// TIA Portal V20 export
// export: Created 2025-12-01T14:57:40.422597Z, ExportSetting None, DisplayName Totally Integrated Automation Portal, DisplayVersion V20 Update 3, DisplayName TIA Portal Openness, DisplayVersion V20 Update 3, DisplayName TIA Portal Version Control Interface, DisplayVersion V20 Update 3, DisplayName STEP 7 Professional, DisplayVersion V20 Update 3, DisplayName STEP 7 Safety, DisplayVersion V20 Update 2, DisplayName WinCC Basic/Comfort/Advanced, DisplayVersion V20 Update 3, DisplayName WinCC Professional, DisplayVersion V20 Update 3, DisplayName WinCC Unified, DisplayVersion V20 Update 3
FUNCTION_BLOCK "FB290_M_CIMCORP_Carga"   // FB290, LAD
TITLE = M_TRANSLO_CS_CARGA_E1_S0
{ S7_Optimized_Access := 'FALSE' }
AUTHOR : CIMCORP
NAME : 20170822
VERSION : 3.5
// stored: AutoNumber false, SetENOAutomatically false
   VAR_INPUT
      Mesa : UInt;   // Mesa de la FB
      Error_Tx : Bool;   // Error en el Tx
      EnTension : Bool;   // Existe Tension en la Mesa
      Termico_Tx : Bool;   // Proteccion del Tx
      pHsMx_1 : Bool;   // pHs 1 de la Mesa
      pHsMx_2 : Bool;   // pHs 2 de la Mesa
      pHsMx_Seg : Bool;   // pHs Seguridad de la Mesa
      Avance_Tx : Bool;   // Avance del Tx
      CIMCORP_MoveOK : Bool;   // CIMCORP >> Move OK
      CIMCORP_Stop : Bool;   // CIMCORP >> Stop
      Centrador_OUT : Bool;   // CENTRADOR >> OUT - Fuera
      Centrador_IN { ExternalAccessible := 'False'; ExternalVisible := 'False'; ExternalWritable := 'False'} : Bool;   // CENTRADOR >> IN - Dentro
      Centrador_EnMovimiento : Bool;   // CENTRADOR >> En Movimiento
      MAnt_CajaPequena : Bool;   // E1 >> Mesa Anterior Caja Pequeña
      MAnt_DescargaAct : Bool;   // E1 >> Mesa Anterior DescargaAct
      AVTF_MAnt_Mx : Bool;   // E1 >> Mesa Anterior AVTF
      P_Mens_MAnt_Mx : Bool;   // E1 >> Mesa Anterior P_Mens
      Mx_ControlUTs : Bool;   // Config >> Control de UT en Mesa
      Mx_VelocidadLenta_In : Bool;   // Forzar a Velociada Lenta
      F_EnvMens_Mx : Bool;   // Fin de Envio de Mensaje
      OrdSal_S00 : Bool;   // Orden de Salida por S0
      V_CNT_pHsMx : Int := 400;   // Valor de Presencia
      V_CNTSeg_pHsMx : Int := 2000;   // Valor de Seguriadad para Presencia
      V_CNT_PasoLenta : Int := 2000;   // Valor de Paso a Lenta
      V_TOut_Tx_Mx : Int := 15000;   // TimeOut de Entrada por E1
      V_TOut_Centrador : Int := 5000;   // TimeOut del Centrador
      V_TOut_Horquillado : Int := 10000;   // TimeOut de Horquillado
      V_CNT_PerdidapHs : Int := 1000;   // CNT de Perdida de pHs
      V_CNT_Posicionado : Int := 1000;   // CNT de Posicionado Simple
      V_CNT_CargaCompactada : Int := 1000;   // CNT de Carga Compactada
   END_VAR
   VAR_OUTPUT
      P_EnvMens_PMx : Bool;   // Permiso de Enviar Mensaje de Presencia
      P_EnvMens_AMx : Bool;   // Permiso de Enviar Mensaje de Ausencia
      P_RecepOK_Mx : Bool;   // Recepcion OK
      PTF_MAnt_Mx : Bool;   // E1 >> Mesa Anterior PTF
      FTF_MAnt_Mx : Bool;   // E1 >> Mesa Anterior FTF
   END_VAR
   VAR
      Mx_ET00 : Bool;
      Mx_ET01 : Bool;
      Mx_ET02 : Bool;
      Mx_ET07_1PRE : Bool;
      Mx_ET07_1FIN : Bool;
      Mx_ET07_2PRE : Bool;
      Mx_ET07_2FIN : Bool;
      Mx_ET08 : Bool;
      Mx_ET09 : Bool;
      Mx_ET10Previo : Bool;
      Mx_ET10 : Bool;
      Mx_ET11 : Bool;
      Mx_ET12 : Bool;
      Mx_ET110 : Bool;
      Mx_ET111 : Bool;
      Mx_ET02ESPERA : Bool;
      Mx_ET50 : Bool;
      Mx_ET51 : Bool;
      Mx_ET52 : Bool;
      MX_ET150 : Bool;
      Mx_ET151 : Bool;
      Mx_EnResetDoblePres : Bool;   // Config >> En Reset Doble Presencia
      CIMCORP_OK : Bool;   // CIMCORP >> Esta En Marcha
      SinUTs_EnMesa : Bool;   // Control UTs En Mesa >> Sin UTs
      DoblePeque_EnMesa : Bool;   // Control UTs En Mesa >> Caja Doble Pequeña
      UT01Peque_EnMesa : Bool;   // Control UTs En Mesa >> UT01 Caja Pequeña
      UT02Peque_EnMesa : Bool;   // Control UTs En Mesa >> UT02 Caja Pequeña
      OrdSalida_OK : Bool;   // Control UTs En Mesa >> Validar Orden de Salida
      EntrandoDobleCaja : Bool;   // Interna >> Entrando Doble Caja
      SalidaDobleCaja : Bool;   // Interna >> Salida de Caja Grande o Dos Pequeñas
      SalidaSimpleCaja : Bool;   // Interna >> Salida de Caja pequeña
      CargaCompactada : Bool;   // Interna >> Carga Compactada
      MemoriaCentrador_IN : Bool;   // Interna >> Memoria para la Señal de Centrador IN
      ProtocoloIniciado : Bool;   // Iniciado el Envio del Mensaje de Presencia
      CNT_pHsMx { S7_SetPoint := 'True'} : "FB910_CNT_UHS";   // CNT de la Presencia
      CNTSeg_pHsMx { S7_SetPoint := 'True'} : "FB910_CNT_UHS";   // CNT de Seguridad de la Presencia
      TMP_EnTension { S7_SetPoint := 'True'} : "FB910_CNT_UHS";
      TOut_Av_Tx { ExternalWritable := 'False'; S7_SetPoint := 'True'} : "FB910_CNT_UHS";   // Time Out de Entrada de E1
      TOut_SacarCentrador { S7_SetPoint := 'True'} : "FB910_CNT_UHS";
      TOut_RecogerCentrador { S7_SetPoint := 'True'} : "FB910_CNT_UHS";
      TOut_Horquillado { S7_SetPoint := 'True'} : "FB910_CNT_UHS";
      CNT_PerdidapHs { S7_SetPoint := 'True'} : "FB910_CNT_UHS";   // CNT de Perdida de pHs
      CNT_Posicionado { S7_SetPoint := 'True'} : "FB910_CNT_UHS";   // CNT de Posicionado Simple
      CNT_CargaCompactada { S7_SetPoint := 'True'} : "FB910_CNT_UHS";   // CNT de Carga Compactada
      STAT_EnvMens_PMx : Bool;   // Interna >> Envio del Mensaje de Presencia
      STAT_EnvMens_AMx : Bool;   // Interna >> Envio de Mensaje de Ausencia
      STAT_FTF_MAnt_Mx : Bool;   // Interna >> FTF de MAnt >> Mx
      MA_LoadOK : Bool;
      MA_SacarCentrador : Bool;
      MA_RecogerCentrador : Bool;
   END_VAR
   VAR_TEMP
      EstadoZona : "EstadoZona";   // Estado de Zona de la Mesa
      EstadoVI : "EstadosMesa";   // Estado del Vehiculo Inteliguente de la Mesa
      ConfigFB : "UDT_ConfigFB";   // Configuracion de la FB de la Mesa
      Aux_ET00 : Bool;
   END_VAR
BEGIN

REGION Network 1: CONFIGURACIONES ESPECIALES DE LA FB
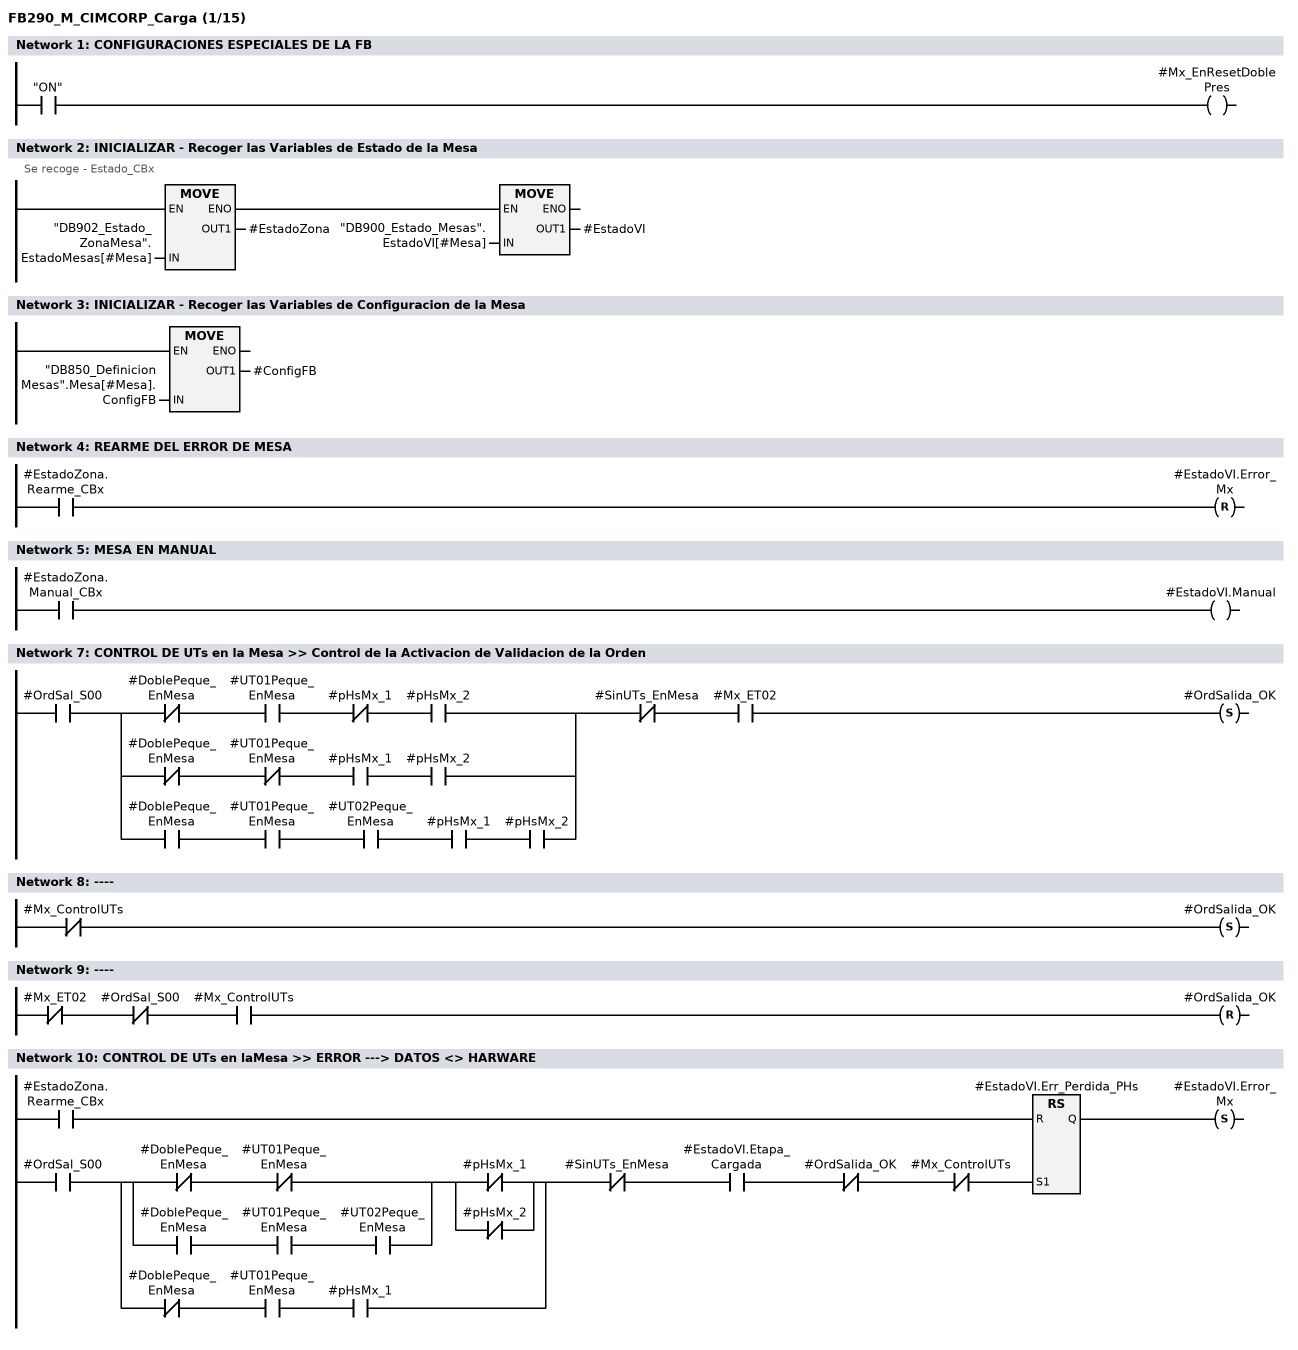
   RUNG wire#powerrail
      Contact( "ON" )
      Coil( #Mx_EnResetDoblePres )
   END_RUNG
   // the same network as SCL:
   #Mx_EnResetDoblePres := "ON";
END_REGION

REGION Network 2: INICIALIZAR - Recoger las Variables de Estado de la Mesa
   // Se recoge - Estado_CBx
   RUNG wire#powerrail
      Move(in := "DB902_Estado_ZonaMesa".EstadoMesas[#Mesa], out1 => #EstadoZona)
      Move(in := "DB900_Estado_Mesas".EstadoVI[#Mesa], out1 => #EstadoVI)
   END_RUNG
   // the same network as SCL:
   #EstadoZona := "DB902_Estado_ZonaMesa".EstadoMesas[#Mesa];
   #EstadoVI := "DB900_Estado_Mesas".EstadoVI[#Mesa];
END_REGION

REGION Network 3: INICIALIZAR - Recoger las Variables de Configuracion de la Mesa
   RUNG wire#powerrail
      Move(in := "DB850_DefinicionMesas".Mesa[#Mesa].ConfigFB, out1 => #ConfigFB)
   END_RUNG
   // the same network as SCL:
   #ConfigFB := "DB850_DefinicionMesas".Mesa[#Mesa].ConfigFB;
END_REGION

REGION Network 4: REARME DEL ERROR DE MESA
   RUNG wire#powerrail
      Contact( #EstadoZona.Rearme_CBx )
      R_Coil( #EstadoVI.Error_Mx )
   END_RUNG
   // the same network as SCL:
   IF #EstadoZona.Rearme_CBx THEN #EstadoVI.Error_Mx := FALSE; END_IF;
END_REGION

REGION Network 5: MESA EN MANUAL
   RUNG wire#powerrail
      Contact( #EstadoZona.Manual_CBx )
      Coil( #EstadoVI.Manual )
   END_RUNG
   // the same network as SCL:
   #EstadoVI.Manual := #EstadoZona.Manual_CBx;
END_REGION

NETWORK
TITLE = CONTROL DE UTs en la Mesa >> Recoger datos de las UTs de la Mesa
//////////////////////////////////////////////////////////////////////////////////
/// Recoger datos de las UTs de la Mesa

      CALL  "FC870_MesaSinUT"
      ( Mesa  := #Mesa,
        SinUT := #SinUTs_EnMesa
      );

      CALL  "FC777_TipoCajaPlastico_EnMesa"
      ( Mesa           := #Mesa,
        DosCajas       := #DoblePeque_EnMesa,
        CajaPeque_UT01 := #UT01Peque_EnMesa,
        CajaPeque_UT02 := #UT02Peque_EnMesa
      );



REGION Network 7: CONTROL DE UTs en la Mesa >> Control de la Activacion de Validacion de la Orden
   RUNG wire#powerrail
      Contact( #OrdSal_S00 )
      wire#w1
      I_Contact( #DoblePeque_EnMesa )
      Contact( #UT01Peque_EnMesa )
      I_Contact( #pHsMx_1 )
      Contact( #pHsMx_2 )
      wire#w2
      I_Contact( #SinUTs_EnMesa )
      Contact( #Mx_ET02 )
      S_Coil( #OrdSalida_OK )
   END_RUNG
   RUNG wire#w1
      I_Contact( #DoblePeque_EnMesa )
      I_Contact( #UT01Peque_EnMesa )
      Contact( #pHsMx_1 )
      Contact( #pHsMx_2 )
   END_RUNG wire#w2
   RUNG wire#w1
      Contact( #DoblePeque_EnMesa )
      Contact( #UT01Peque_EnMesa )
      Contact( #UT02Peque_EnMesa )
      Contact( #pHsMx_1 )
      Contact( #pHsMx_2 )
   END_RUNG wire#w2
   // the same network as SCL:
   IF #OrdSal_S00 AND ((NOT #DoblePeque_EnMesa AND #UT01Peque_EnMesa AND NOT #pHsMx_1 AND #pHsMx_2) OR (NOT #DoblePeque_EnMesa AND NOT #UT01Peque_EnMesa AND #pHsMx_1 AND #pHsMx_2) OR (#DoblePeque_EnMesa AND #UT01Peque_EnMesa AND #UT02Peque_EnMesa AND #pHsMx_1 AND #pHsMx_2)) AND NOT #SinUTs_EnMesa AND #Mx_ET02 THEN
       #OrdSalida_OK := TRUE;
   END_IF;
END_REGION

REGION Network 8: ----
   RUNG wire#powerrail
      I_Contact( #Mx_ControlUTs )
      S_Coil( #OrdSalida_OK )
   END_RUNG
   // the same network as SCL:
   IF NOT #Mx_ControlUTs THEN #OrdSalida_OK := TRUE; END_IF;
END_REGION

REGION Network 9: ----
   RUNG wire#powerrail
      I_Contact( #Mx_ET02 )
      I_Contact( #OrdSal_S00 )
      Contact( #Mx_ControlUTs )
      R_Coil( #OrdSalida_OK )
   END_RUNG
   // the same network as SCL:
   IF NOT #Mx_ET02 AND NOT #OrdSal_S00 AND #Mx_ControlUTs THEN #OrdSalida_OK := FALSE; END_IF;
END_REGION

REGION Network 10: CONTROL DE UTs en laMesa >> ERROR ---> DATOS <> HARWARE
   RUNG wire#powerrail
      Contact( #EstadoZona.Rearme_CBx )
      S_RS(operand := #EstadoVI.Err_Perdida_PHs, s1 := wire#w4)
      S_Coil( #EstadoVI.Error_Mx )
   END_RUNG
   RUNG wire#powerrail
      Contact( #OrdSal_S00 )
      wire#w1
      I_Contact( #DoblePeque_EnMesa )
      I_Contact( #UT01Peque_EnMesa )
      wire#w2
      I_Contact( #pHsMx_1 )
      wire#w3
      I_Contact( #SinUTs_EnMesa )
      Contact( #EstadoVI.Etapa_Cargada )
      I_Contact( #OrdSalida_OK )
      I_Contact( #Mx_ControlUTs )
   END_RUNG wire#w4
   RUNG wire#w1
      Contact( #DoblePeque_EnMesa )
      Contact( #UT01Peque_EnMesa )
      Contact( #UT02Peque_EnMesa )
   END_RUNG wire#w2
   RUNG wire#w2
      I_Contact( #pHsMx_2 )
   END_RUNG wire#w3
   RUNG wire#w1
      I_Contact( #DoblePeque_EnMesa )
      Contact( #UT01Peque_EnMesa )
      Contact( #pHsMx_1 )
   END_RUNG wire#w3
   // the same network as SCL:
   IF #EstadoZona.Rearme_CBx THEN
       #EstadoVI.Err_Perdida_PHs := FALSE;   // RS flip-flop
   END_IF;
   IF #OrdSal_S00 AND ((((NOT #DoblePeque_EnMesa AND NOT #UT01Peque_EnMesa) OR (#DoblePeque_EnMesa AND #UT01Peque_EnMesa AND #UT02Peque_EnMesa)) AND (NOT #pHsMx_1 OR NOT #pHsMx_2)) OR (NOT #DoblePeque_EnMesa AND #UT01Peque_EnMesa AND #pHsMx_1)) AND NOT #SinUTs_EnMesa AND #EstadoVI.Etapa_Cargada AND NOT #OrdSalida_OK AND NOT #Mx_ControlUTs THEN
       #EstadoVI.Err_Perdida_PHs := TRUE;
   END_IF;
   IF #EstadoVI.Err_Perdida_PHs THEN #EstadoVI.Error_Mx := TRUE; END_IF;
END_REGION

REGION Network 11: VARIABLES AUXILIARES - CONTROL DE CIMCORP
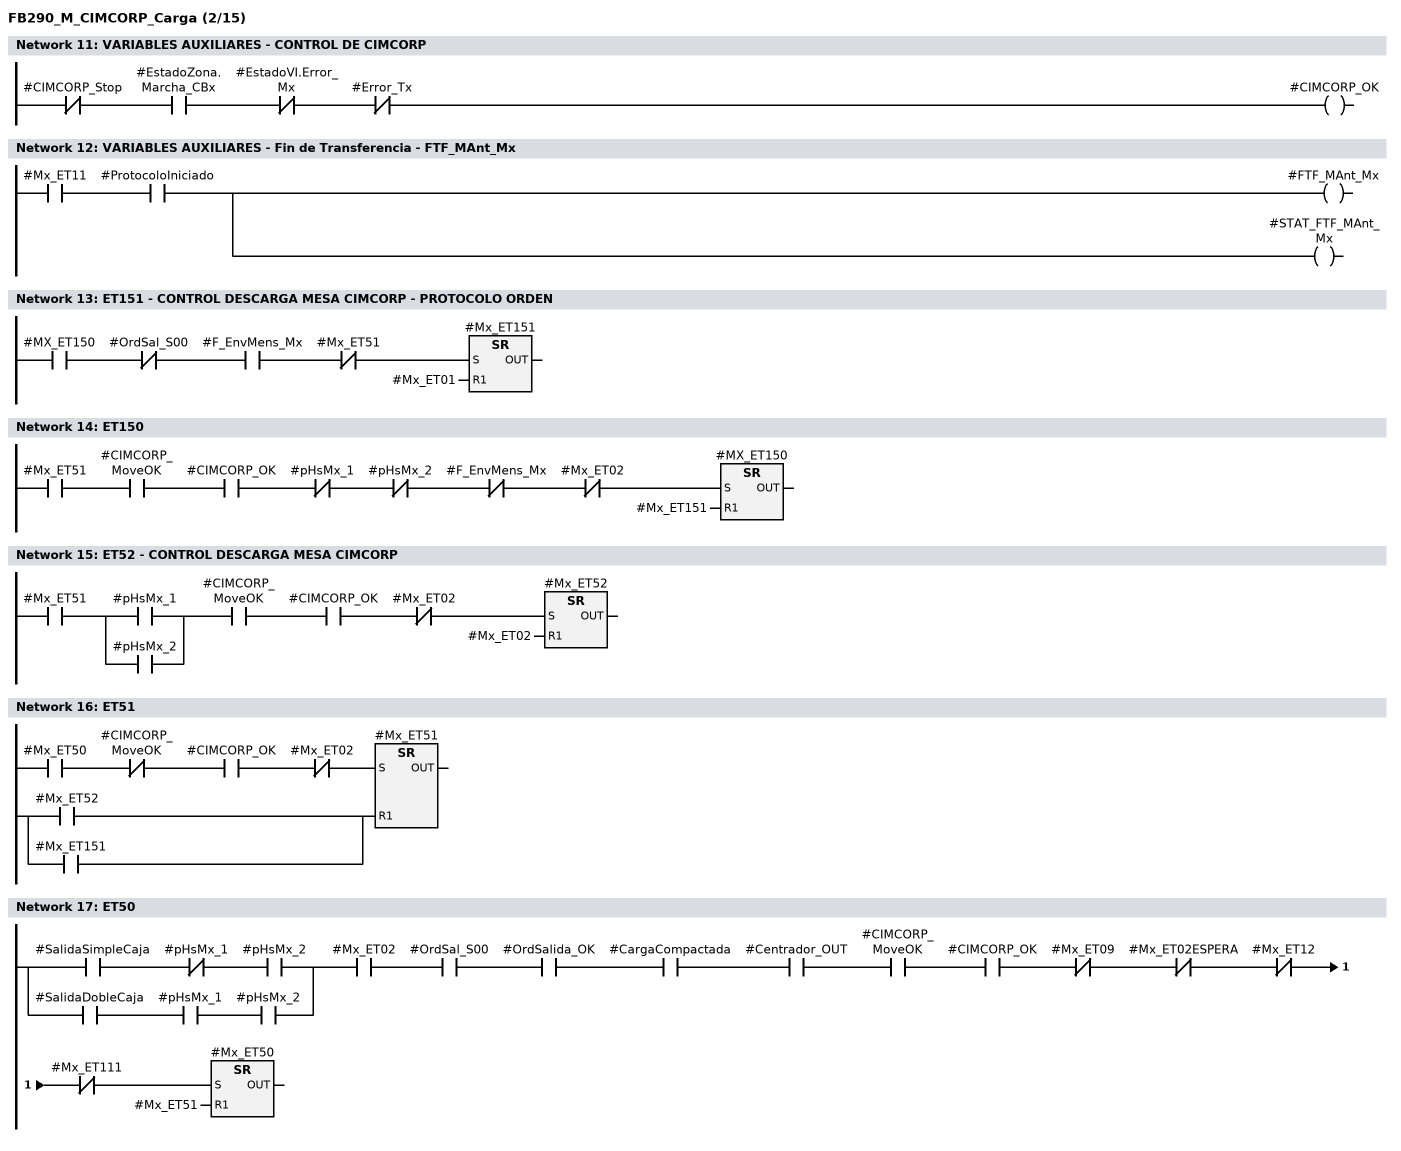
   RUNG wire#powerrail
      I_Contact( #CIMCORP_Stop )
      Contact( #EstadoZona.Marcha_CBx )
      I_Contact( #EstadoVI.Error_Mx )
      I_Contact( #Error_Tx )
      Coil( #CIMCORP_OK )
   END_RUNG
   // the same network as SCL:
   #CIMCORP_OK := NOT #CIMCORP_Stop AND #EstadoZona.Marcha_CBx AND NOT #EstadoVI.Error_Mx AND NOT #Error_Tx;
END_REGION

REGION Network 12: VARIABLES AUXILIARES - Fin de Transferencia - FTF_MAnt_Mx
   RUNG wire#powerrail
      Contact( #Mx_ET11 )
      Contact( #ProtocoloIniciado )
      wire#w1
      Coil( #FTF_MAnt_Mx )
   END_RUNG
   RUNG wire#w1
      Coil( #STAT_FTF_MAnt_Mx )
   END_RUNG
   // the same network as SCL:
   #FTF_MAnt_Mx := #Mx_ET11 AND #ProtocoloIniciado;
   #STAT_FTF_MAnt_Mx := #FTF_MAnt_Mx;
END_REGION

REGION Network 13: ET151 - CONTROL DESCARGA MESA CIMCORP - PROTOCOLO ORDEN
   RUNG wire#powerrail
      Contact( #MX_ET150 )
      I_Contact( #OrdSal_S00 )
      Contact( #F_EnvMens_Mx )
      I_Contact( #Mx_ET51 )
      S_SR(operand := #Mx_ET151, r1 := #Mx_ET01)
   END_RUNG
   // the same network as SCL:
   IF #MX_ET150 AND NOT #OrdSal_S00 AND #F_EnvMens_Mx AND NOT #Mx_ET51 THEN
       #Mx_ET151 := TRUE;   // SR flip-flop
   END_IF;
   IF #Mx_ET01 THEN #Mx_ET151 := FALSE; END_IF;
END_REGION

REGION Network 14: ET150
   RUNG wire#powerrail
      Contact( #Mx_ET51 )
      Contact( #CIMCORP_MoveOK )
      Contact( #CIMCORP_OK )
      I_Contact( #pHsMx_1 )
      I_Contact( #pHsMx_2 )
      I_Contact( #F_EnvMens_Mx )
      I_Contact( #Mx_ET02 )
      S_SR(operand := #MX_ET150, r1 := #Mx_ET151)
   END_RUNG
   // the same network as SCL:
   IF #Mx_ET51 AND #CIMCORP_MoveOK AND #CIMCORP_OK AND NOT #pHsMx_1 AND NOT #pHsMx_2 AND NOT #F_EnvMens_Mx AND NOT #Mx_ET02 THEN
       #MX_ET150 := TRUE;   // SR flip-flop
   END_IF;
   IF #Mx_ET151 THEN #MX_ET150 := FALSE; END_IF;
END_REGION

REGION Network 15: ET52 - CONTROL DESCARGA MESA CIMCORP
   RUNG wire#powerrail
      Contact( #Mx_ET51 )
      wire#w1
      Contact( #pHsMx_1 )
      wire#w2
      Contact( #CIMCORP_MoveOK )
      Contact( #CIMCORP_OK )
      I_Contact( #Mx_ET02 )
      S_SR(operand := #Mx_ET52, r1 := #Mx_ET02)
   END_RUNG
   RUNG wire#w1
      Contact( #pHsMx_2 )
   END_RUNG wire#w2
   // the same network as SCL:
   IF #Mx_ET51 AND (#pHsMx_1 OR #pHsMx_2) AND #CIMCORP_MoveOK AND #CIMCORP_OK AND NOT #Mx_ET02 THEN
       #Mx_ET52 := TRUE;   // SR flip-flop
   END_IF;
   IF #Mx_ET02 THEN #Mx_ET52 := FALSE; END_IF;
END_REGION

REGION Network 16: ET51
   RUNG wire#powerrail
      Contact( #Mx_ET50 )
      I_Contact( #CIMCORP_MoveOK )
      Contact( #CIMCORP_OK )
      I_Contact( #Mx_ET02 )
      S_SR(operand := #Mx_ET51, r1 := wire#w1)
   END_RUNG
   RUNG wire#powerrail
      Contact( #Mx_ET52 )
   END_RUNG wire#w1
   RUNG wire#powerrail
      Contact( #Mx_ET151 )
   END_RUNG wire#w1
   // the same network as SCL:
   IF #Mx_ET50 AND NOT #CIMCORP_MoveOK AND #CIMCORP_OK AND NOT #Mx_ET02 THEN
       #Mx_ET51 := TRUE;   // SR flip-flop
   END_IF;
   IF #Mx_ET52 OR #Mx_ET151 THEN #Mx_ET51 := FALSE; END_IF;
END_REGION

REGION Network 17: ET50
   RUNG wire#powerrail
      Contact( #SalidaSimpleCaja )
      I_Contact( #pHsMx_1 )
      Contact( #pHsMx_2 )
      wire#w1
      Contact( #Mx_ET02 )
      Contact( #OrdSal_S00 )
      Contact( #OrdSalida_OK )
      Contact( #CargaCompactada )
      Contact( #Centrador_OUT )
      Contact( #CIMCORP_MoveOK )
      Contact( #CIMCORP_OK )
      I_Contact( #Mx_ET09 )
      I_Contact( #Mx_ET02ESPERA )
      I_Contact( #Mx_ET12 )
      I_Contact( #Mx_ET111 )
      S_SR(operand := #Mx_ET50, r1 := #Mx_ET51)
   END_RUNG
   RUNG wire#powerrail
      Contact( #SalidaDobleCaja )
      Contact( #pHsMx_1 )
      Contact( #pHsMx_2 )
   END_RUNG wire#w1
   // the same network as SCL:
   IF ((#SalidaSimpleCaja AND NOT #pHsMx_1 AND #pHsMx_2) OR (#SalidaDobleCaja AND #pHsMx_1 AND #pHsMx_2)) AND #Mx_ET02 AND #OrdSal_S00 AND #OrdSalida_OK AND #CargaCompactada AND #Centrador_OUT AND #CIMCORP_MoveOK AND #CIMCORP_OK AND NOT #Mx_ET09 AND NOT #Mx_ET02ESPERA AND NOT #Mx_ET12 AND NOT #Mx_ET111 THEN
       #Mx_ET50 := TRUE;   // SR flip-flop
   END_IF;
   IF #Mx_ET51 THEN #Mx_ET50 := FALSE; END_IF;
END_REGION

REGION Network 18: ET02 - ESTADO REPOSO CARGADA
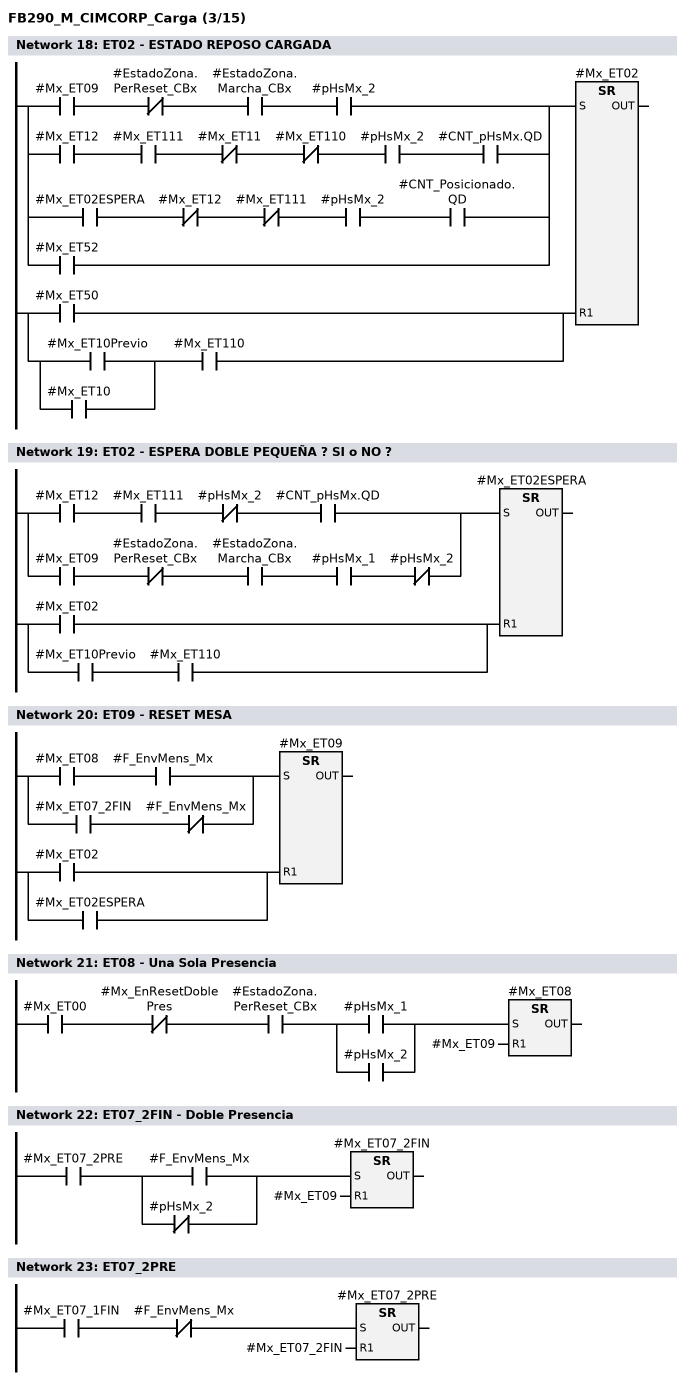
   RUNG wire#powerrail
      Contact( #Mx_ET09 )
      I_Contact( #EstadoZona.PerReset_CBx )
      Contact( #EstadoZona.Marcha_CBx )
      Contact( #pHsMx_2 )
      wire#w1
      S_SR(operand := #Mx_ET02, r1 := wire#w3)
   END_RUNG
   RUNG wire#powerrail
      Contact( #Mx_ET12 )
      Contact( #Mx_ET111 )
      I_Contact( #Mx_ET11 )
      I_Contact( #Mx_ET110 )
      Contact( #pHsMx_2 )
      Contact( #CNT_pHsMx.QD )
   END_RUNG wire#w1
   RUNG wire#powerrail
      Contact( #Mx_ET02ESPERA )
      I_Contact( #Mx_ET12 )
      I_Contact( #Mx_ET111 )
      Contact( #pHsMx_2 )
      Contact( #CNT_Posicionado.QD )
   END_RUNG wire#w1
   RUNG wire#powerrail
      Contact( #Mx_ET52 )
   END_RUNG wire#w1
   RUNG wire#powerrail
      Contact( #Mx_ET50 )
   END_RUNG wire#w3
   RUNG wire#powerrail
      Contact( #Mx_ET10Previo )
      wire#w2
      Contact( #Mx_ET110 )
   END_RUNG wire#w3
   RUNG wire#powerrail
      Contact( #Mx_ET10 )
   END_RUNG wire#w2
   // the same network as SCL:
   IF (#Mx_ET09 AND NOT #EstadoZona.PerReset_CBx AND #EstadoZona.Marcha_CBx AND #pHsMx_2) OR (#Mx_ET12 AND #Mx_ET111 AND NOT #Mx_ET11 AND NOT #Mx_ET110 AND #pHsMx_2 AND #CNT_pHsMx.QD) OR (#Mx_ET02ESPERA AND NOT #Mx_ET12 AND NOT #Mx_ET111 AND #pHsMx_2 AND #CNT_Posicionado.QD) OR #Mx_ET52 THEN
       #Mx_ET02 := TRUE;   // SR flip-flop
   END_IF;
   IF #Mx_ET50 OR ((#Mx_ET10Previo OR #Mx_ET10) AND #Mx_ET110) THEN #Mx_ET02 := FALSE; END_IF;
END_REGION

REGION Network 19: ET02 - ESPERA DOBLE PEQUEÑA ? SI o NO ?
   RUNG wire#powerrail
      Contact( #Mx_ET12 )
      Contact( #Mx_ET111 )
      I_Contact( #pHsMx_2 )
      Contact( #CNT_pHsMx.QD )
      wire#w1
      S_SR(operand := #Mx_ET02ESPERA, r1 := wire#w2)
   END_RUNG
   RUNG wire#powerrail
      Contact( #Mx_ET09 )
      I_Contact( #EstadoZona.PerReset_CBx )
      Contact( #EstadoZona.Marcha_CBx )
      Contact( #pHsMx_1 )
      I_Contact( #pHsMx_2 )
   END_RUNG wire#w1
   RUNG wire#powerrail
      Contact( #Mx_ET02 )
   END_RUNG wire#w2
   RUNG wire#powerrail
      Contact( #Mx_ET10Previo )
      Contact( #Mx_ET110 )
   END_RUNG wire#w2
   // the same network as SCL:
   IF (#Mx_ET12 AND #Mx_ET111 AND NOT #pHsMx_2 AND #CNT_pHsMx.QD) OR (#Mx_ET09 AND NOT #EstadoZona.PerReset_CBx AND #EstadoZona.Marcha_CBx AND #pHsMx_1 AND NOT #pHsMx_2) THEN
       #Mx_ET02ESPERA := TRUE;   // SR flip-flop
   END_IF;
   IF #Mx_ET02 OR (#Mx_ET10Previo AND #Mx_ET110) THEN #Mx_ET02ESPERA := FALSE; END_IF;
END_REGION

REGION Network 20: ET09 - RESET MESA
   RUNG wire#powerrail
      Contact( #Mx_ET08 )
      Contact( #F_EnvMens_Mx )
      wire#w1
      S_SR(operand := #Mx_ET09, r1 := wire#w2)
   END_RUNG
   RUNG wire#powerrail
      Contact( #Mx_ET07_2FIN )
      I_Contact( #F_EnvMens_Mx )
   END_RUNG wire#w1
   RUNG wire#powerrail
      Contact( #Mx_ET02 )
   END_RUNG wire#w2
   RUNG wire#powerrail
      Contact( #Mx_ET02ESPERA )
   END_RUNG wire#w2
   // the same network as SCL:
   IF (#Mx_ET08 AND #F_EnvMens_Mx) OR (#Mx_ET07_2FIN AND NOT #F_EnvMens_Mx) THEN
       #Mx_ET09 := TRUE;   // SR flip-flop
   END_IF;
   IF #Mx_ET02 OR #Mx_ET02ESPERA THEN #Mx_ET09 := FALSE; END_IF;
END_REGION

REGION Network 21: ET08 - Una Sola Presencia
   RUNG wire#powerrail
      Contact( #Mx_ET00 )
      I_Contact( #Mx_EnResetDoblePres )
      Contact( #EstadoZona.PerReset_CBx )
      wire#w1
      Contact( #pHsMx_1 )
      wire#w2
      S_SR(operand := #Mx_ET08, r1 := #Mx_ET09)
   END_RUNG
   RUNG wire#w1
      Contact( #pHsMx_2 )
   END_RUNG wire#w2
   // the same network as SCL:
   IF #Mx_ET00 AND NOT #Mx_EnResetDoblePres AND #EstadoZona.PerReset_CBx AND (#pHsMx_1 OR #pHsMx_2) THEN
       #Mx_ET08 := TRUE;   // SR flip-flop
   END_IF;
   IF #Mx_ET09 THEN #Mx_ET08 := FALSE; END_IF;
END_REGION

REGION Network 22: ET07_2FIN - Doble Presencia
   RUNG wire#powerrail
      Contact( #Mx_ET07_2PRE )
      wire#w1
      Contact( #F_EnvMens_Mx )
      wire#w2
      S_SR(operand := #Mx_ET07_2FIN, r1 := #Mx_ET09)
   END_RUNG
   RUNG wire#w1
      I_Contact( #pHsMx_2 )
   END_RUNG wire#w2
   // the same network as SCL:
   IF #Mx_ET07_2PRE AND (#F_EnvMens_Mx OR NOT #pHsMx_2) THEN
       #Mx_ET07_2FIN := TRUE;   // SR flip-flop
   END_IF;
   IF #Mx_ET09 THEN #Mx_ET07_2FIN := FALSE; END_IF;
END_REGION

REGION Network 23: ET07_2PRE
   RUNG wire#powerrail
      Contact( #Mx_ET07_1FIN )
      I_Contact( #F_EnvMens_Mx )
      S_SR(operand := #Mx_ET07_2PRE, r1 := #Mx_ET07_2FIN)
   END_RUNG
   // the same network as SCL:
   IF #Mx_ET07_1FIN AND NOT #F_EnvMens_Mx THEN
       #Mx_ET07_2PRE := TRUE;   // SR flip-flop
   END_IF;
   IF #Mx_ET07_2FIN THEN #Mx_ET07_2PRE := FALSE; END_IF;
END_REGION

REGION Network 24: ET07_1FIN
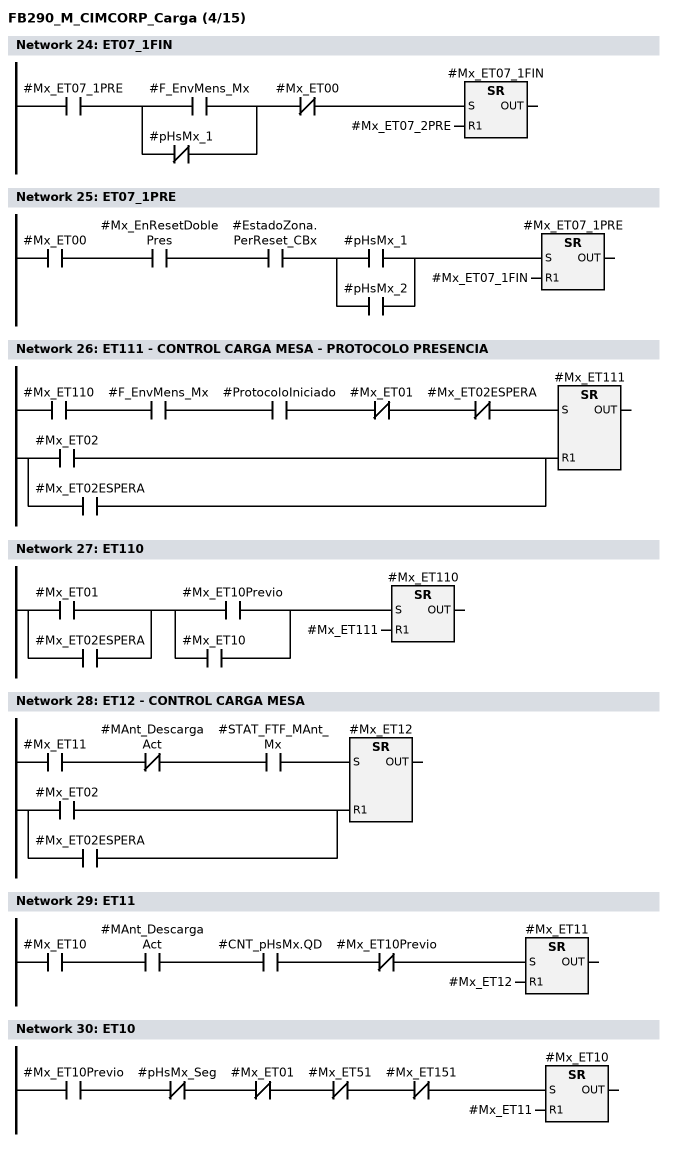
   RUNG wire#powerrail
      Contact( #Mx_ET07_1PRE )
      wire#w1
      Contact( #F_EnvMens_Mx )
      wire#w2
      I_Contact( #Mx_ET00 )
      S_SR(operand := #Mx_ET07_1FIN, r1 := #Mx_ET07_2PRE)
   END_RUNG
   RUNG wire#w1
      I_Contact( #pHsMx_1 )
   END_RUNG wire#w2
   // the same network as SCL:
   IF #Mx_ET07_1PRE AND (#F_EnvMens_Mx OR NOT #pHsMx_1) AND NOT #Mx_ET00 THEN
       #Mx_ET07_1FIN := TRUE;   // SR flip-flop
   END_IF;
   IF #Mx_ET07_2PRE THEN #Mx_ET07_1FIN := FALSE; END_IF;
END_REGION

REGION Network 25: ET07_1PRE
   RUNG wire#powerrail
      Contact( #Mx_ET00 )
      Contact( #Mx_EnResetDoblePres )
      Contact( #EstadoZona.PerReset_CBx )
      wire#w1
      Contact( #pHsMx_1 )
      wire#w2
      S_SR(operand := #Mx_ET07_1PRE, r1 := #Mx_ET07_1FIN)
   END_RUNG
   RUNG wire#w1
      Contact( #pHsMx_2 )
   END_RUNG wire#w2
   // the same network as SCL:
   IF #Mx_ET00 AND #Mx_EnResetDoblePres AND #EstadoZona.PerReset_CBx AND (#pHsMx_1 OR #pHsMx_2) THEN
       #Mx_ET07_1PRE := TRUE;   // SR flip-flop
   END_IF;
   IF #Mx_ET07_1FIN THEN #Mx_ET07_1PRE := FALSE; END_IF;
END_REGION

REGION Network 26: ET111 - CONTROL CARGA MESA - PROTOCOLO PRESENCIA
   RUNG wire#powerrail
      Contact( #Mx_ET110 )
      Contact( #F_EnvMens_Mx )
      Contact( #ProtocoloIniciado )
      I_Contact( #Mx_ET01 )
      I_Contact( #Mx_ET02ESPERA )
      S_SR(operand := #Mx_ET111, r1 := wire#w1)
   END_RUNG
   RUNG wire#powerrail
      Contact( #Mx_ET02 )
   END_RUNG wire#w1
   RUNG wire#powerrail
      Contact( #Mx_ET02ESPERA )
   END_RUNG wire#w1
   // the same network as SCL:
   IF #Mx_ET110 AND #F_EnvMens_Mx AND #ProtocoloIniciado AND NOT #Mx_ET01 AND NOT #Mx_ET02ESPERA THEN
       #Mx_ET111 := TRUE;   // SR flip-flop
   END_IF;
   IF #Mx_ET02 OR #Mx_ET02ESPERA THEN #Mx_ET111 := FALSE; END_IF;
END_REGION

REGION Network 27: ET110
   RUNG wire#powerrail
      Contact( #Mx_ET01 )
      wire#w1
      Contact( #Mx_ET10Previo )
      wire#w2
      S_SR(operand := #Mx_ET110, r1 := #Mx_ET111)
   END_RUNG
   RUNG wire#powerrail
      Contact( #Mx_ET02ESPERA )
   END_RUNG wire#w1
   RUNG wire#w1
      Contact( #Mx_ET10 )
   END_RUNG wire#w2
   // the same network as SCL:
   IF (#Mx_ET01 OR #Mx_ET02ESPERA) AND (#Mx_ET10Previo OR #Mx_ET10) THEN
       #Mx_ET110 := TRUE;   // SR flip-flop
   END_IF;
   IF #Mx_ET111 THEN #Mx_ET110 := FALSE; END_IF;
END_REGION

REGION Network 28: ET12 - CONTROL CARGA MESA
   RUNG wire#powerrail
      Contact( #Mx_ET11 )
      I_Contact( #MAnt_DescargaAct )
      Contact( #STAT_FTF_MAnt_Mx )
      S_SR(operand := #Mx_ET12, r1 := wire#w1)
   END_RUNG
   RUNG wire#powerrail
      Contact( #Mx_ET02 )
   END_RUNG wire#w1
   RUNG wire#powerrail
      Contact( #Mx_ET02ESPERA )
   END_RUNG wire#w1
   // the same network as SCL:
   IF #Mx_ET11 AND NOT #MAnt_DescargaAct AND #STAT_FTF_MAnt_Mx THEN
       #Mx_ET12 := TRUE;   // SR flip-flop
   END_IF;
   IF #Mx_ET02 OR #Mx_ET02ESPERA THEN #Mx_ET12 := FALSE; END_IF;
END_REGION

REGION Network 29: ET11
   RUNG wire#powerrail
      Contact( #Mx_ET10 )
      Contact( #MAnt_DescargaAct )
      Contact( #CNT_pHsMx.QD )
      I_Contact( #Mx_ET10Previo )
      S_SR(operand := #Mx_ET11, r1 := #Mx_ET12)
   END_RUNG
   // the same network as SCL:
   IF #Mx_ET10 AND #MAnt_DescargaAct AND #CNT_pHsMx.QD AND NOT #Mx_ET10Previo THEN
       #Mx_ET11 := TRUE;   // SR flip-flop
   END_IF;
   IF #Mx_ET12 THEN #Mx_ET11 := FALSE; END_IF;
END_REGION

REGION Network 30: ET10
   RUNG wire#powerrail
      Contact( #Mx_ET10Previo )
      I_Contact( #pHsMx_Seg )
      I_Contact( #Mx_ET01 )
      I_Contact( #Mx_ET51 )
      I_Contact( #Mx_ET151 )
      S_SR(operand := #Mx_ET10, r1 := #Mx_ET11)
   END_RUNG
   // the same network as SCL:
   IF #Mx_ET10Previo AND NOT #pHsMx_Seg AND NOT #Mx_ET01 AND NOT #Mx_ET51 AND NOT #Mx_ET151 THEN
       #Mx_ET10 := TRUE;   // SR flip-flop
   END_IF;
   IF #Mx_ET11 THEN #Mx_ET10 := FALSE; END_IF;
END_REGION

REGION Network 31: ET10Previo - CARGA EN LA pHs de SEG
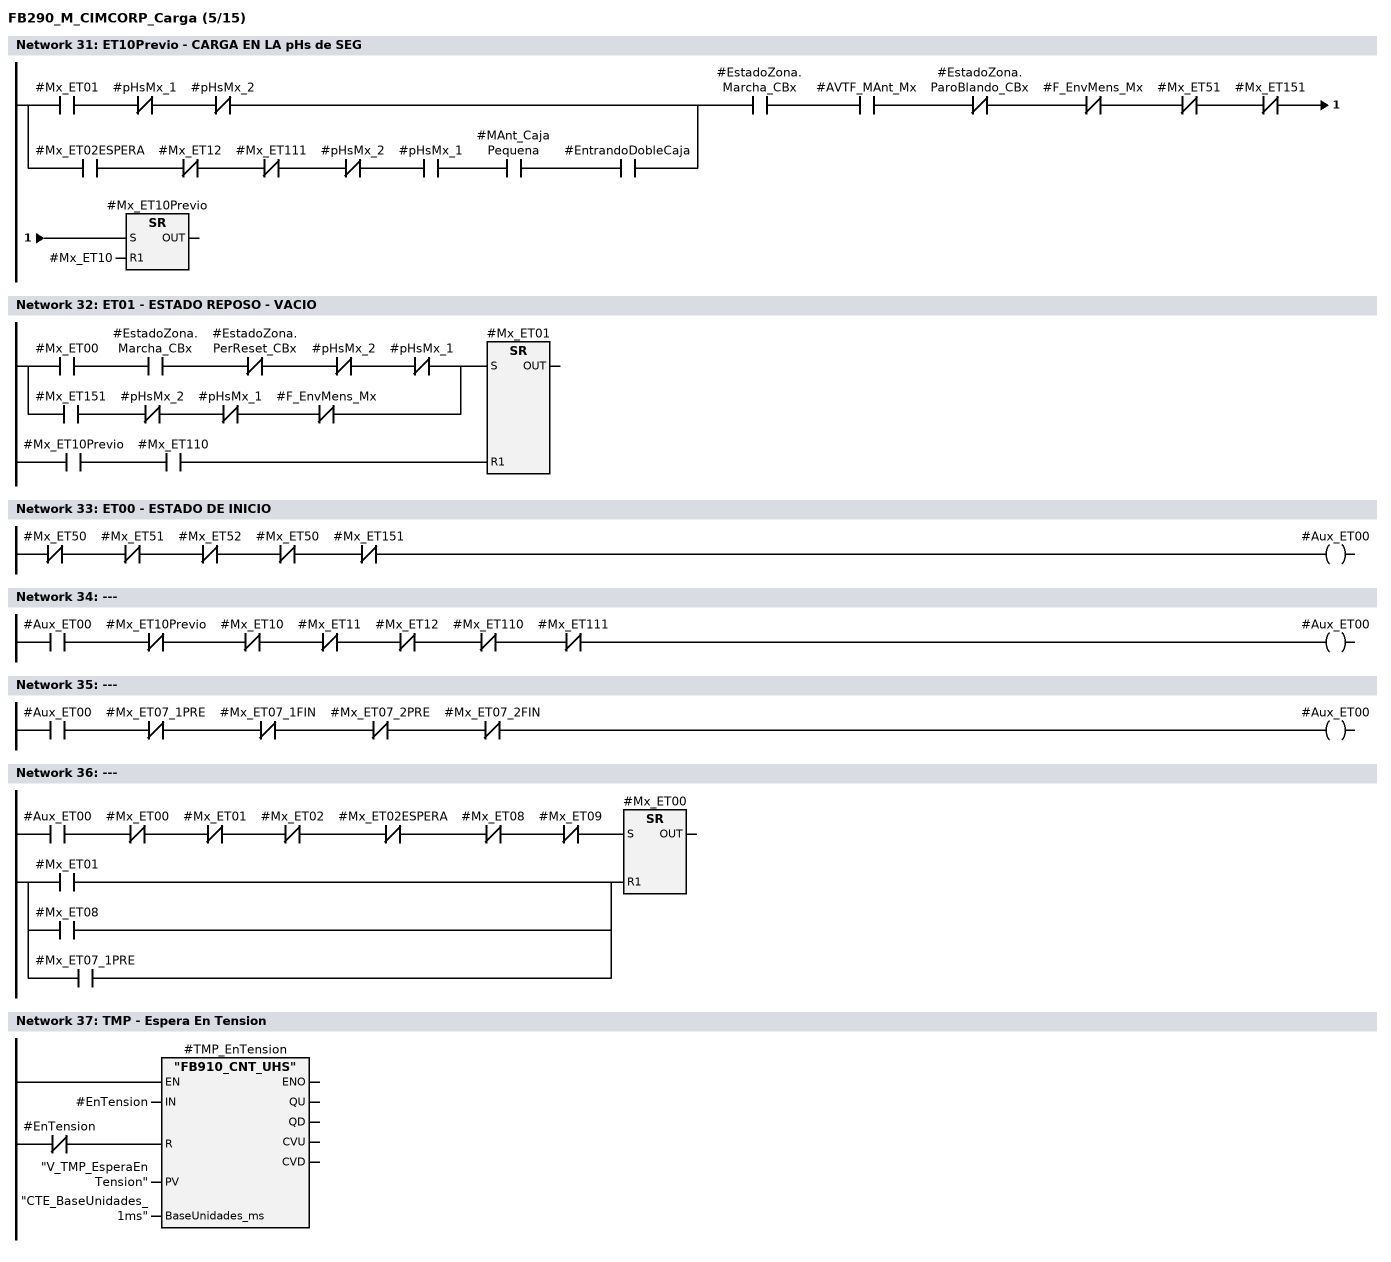
   RUNG wire#powerrail
      Contact( #Mx_ET01 )
      I_Contact( #pHsMx_1 )
      I_Contact( #pHsMx_2 )
      wire#w1
      Contact( #EstadoZona.Marcha_CBx )
      Contact( #AVTF_MAnt_Mx )
      I_Contact( #EstadoZona.ParoBlando_CBx )
      I_Contact( #F_EnvMens_Mx )
      I_Contact( #Mx_ET51 )
      I_Contact( #Mx_ET151 )
      S_SR(operand := #Mx_ET10Previo, r1 := #Mx_ET10)
   END_RUNG
   RUNG wire#powerrail
      Contact( #Mx_ET02ESPERA )
      I_Contact( #Mx_ET12 )
      I_Contact( #Mx_ET111 )
      I_Contact( #pHsMx_2 )
      Contact( #pHsMx_1 )
      Contact( #MAnt_CajaPequena )
      Contact( #EntrandoDobleCaja )
   END_RUNG wire#w1
   // the same network as SCL:
   IF ((#Mx_ET01 AND NOT #pHsMx_1 AND NOT #pHsMx_2) OR (#Mx_ET02ESPERA AND NOT #Mx_ET12 AND NOT #Mx_ET111 AND NOT #pHsMx_2 AND #pHsMx_1 AND #MAnt_CajaPequena AND #EntrandoDobleCaja)) AND #EstadoZona.Marcha_CBx AND #AVTF_MAnt_Mx AND NOT #EstadoZona.ParoBlando_CBx AND NOT #F_EnvMens_Mx AND NOT #Mx_ET51 AND NOT #Mx_ET151 THEN
       #Mx_ET10Previo := TRUE;   // SR flip-flop
   END_IF;
   IF #Mx_ET10 THEN #Mx_ET10Previo := FALSE; END_IF;
END_REGION

REGION Network 32: ET01 - ESTADO REPOSO - VACIO
   RUNG wire#powerrail
      Contact( #Mx_ET00 )
      Contact( #EstadoZona.Marcha_CBx )
      I_Contact( #EstadoZona.PerReset_CBx )
      I_Contact( #pHsMx_2 )
      I_Contact( #pHsMx_1 )
      wire#w1
      S_SR(operand := #Mx_ET01, r1 := wire#w2)
   END_RUNG
   RUNG wire#powerrail
      Contact( #Mx_ET151 )
      I_Contact( #pHsMx_2 )
      I_Contact( #pHsMx_1 )
      I_Contact( #F_EnvMens_Mx )
   END_RUNG wire#w1
   RUNG wire#powerrail
      Contact( #Mx_ET10Previo )
      Contact( #Mx_ET110 )
   END_RUNG wire#w2
   // the same network as SCL:
   IF (#Mx_ET00 AND #EstadoZona.Marcha_CBx AND NOT #EstadoZona.PerReset_CBx AND NOT #pHsMx_2 AND NOT #pHsMx_1) OR (#Mx_ET151 AND NOT #pHsMx_2 AND NOT #pHsMx_1 AND NOT #F_EnvMens_Mx) THEN
       #Mx_ET01 := TRUE;   // SR flip-flop
   END_IF;
   IF #Mx_ET10Previo AND #Mx_ET110 THEN #Mx_ET01 := FALSE; END_IF;
END_REGION

REGION Network 33: ET00 - ESTADO DE INICIO
   RUNG wire#powerrail
      I_Contact( #Mx_ET50 )
      I_Contact( #Mx_ET51 )
      I_Contact( #Mx_ET52 )
      I_Contact( #Mx_ET50 )
      I_Contact( #Mx_ET151 )
      Coil( #Aux_ET00 )
   END_RUNG
   // the same network as SCL:
   #Aux_ET00 := NOT #Mx_ET50 AND NOT #Mx_ET51 AND NOT #Mx_ET52 AND NOT #Mx_ET50 AND NOT #Mx_ET151;
END_REGION

REGION Network 34: ---
   RUNG wire#powerrail
      Contact( #Aux_ET00 )
      I_Contact( #Mx_ET10Previo )
      I_Contact( #Mx_ET10 )
      I_Contact( #Mx_ET11 )
      I_Contact( #Mx_ET12 )
      I_Contact( #Mx_ET110 )
      I_Contact( #Mx_ET111 )
      Coil( #Aux_ET00 )
   END_RUNG
   // the same network as SCL:
   #Aux_ET00 := #Aux_ET00 AND NOT #Mx_ET10Previo AND NOT #Mx_ET10 AND NOT #Mx_ET11 AND NOT #Mx_ET12 AND NOT #Mx_ET110 AND NOT #Mx_ET111;
END_REGION

REGION Network 35: ---
   RUNG wire#powerrail
      Contact( #Aux_ET00 )
      I_Contact( #Mx_ET07_1PRE )
      I_Contact( #Mx_ET07_1FIN )
      I_Contact( #Mx_ET07_2PRE )
      I_Contact( #Mx_ET07_2FIN )
      Coil( #Aux_ET00 )
   END_RUNG
   // the same network as SCL:
   #Aux_ET00 := #Aux_ET00 AND NOT #Mx_ET07_1PRE AND NOT #Mx_ET07_1FIN AND NOT #Mx_ET07_2PRE AND NOT #Mx_ET07_2FIN;
END_REGION

REGION Network 36: ---
   RUNG wire#powerrail
      Contact( #Aux_ET00 )
      I_Contact( #Mx_ET00 )
      I_Contact( #Mx_ET01 )
      I_Contact( #Mx_ET02 )
      I_Contact( #Mx_ET02ESPERA )
      I_Contact( #Mx_ET08 )
      I_Contact( #Mx_ET09 )
      S_SR(operand := #Mx_ET00, r1 := wire#w1)
   END_RUNG
   RUNG wire#powerrail
      Contact( #Mx_ET01 )
   END_RUNG wire#w1
   RUNG wire#powerrail
      Contact( #Mx_ET08 )
   END_RUNG wire#w1
   RUNG wire#powerrail
      Contact( #Mx_ET07_1PRE )
   END_RUNG wire#w1
   // the same network as SCL:
   IF #Aux_ET00 AND NOT #Mx_ET00 AND NOT #Mx_ET01 AND NOT #Mx_ET02 AND NOT #Mx_ET02ESPERA AND NOT #Mx_ET08 AND NOT #Mx_ET09 THEN
       #Mx_ET00 := TRUE;   // SR flip-flop
   END_IF;
   IF #Mx_ET01 OR #Mx_ET08 OR #Mx_ET07_1PRE THEN #Mx_ET00 := FALSE; END_IF;
END_REGION

REGION Network 37: TMP - Espera En Tension
   RUNG wire#powerrail
      #TMP_EnTension(R := wire#w1, IN := #EnTension, PV := "V_TMP_EsperaEnTension", BaseUnidades_ms := "CTE_BaseUnidades_1ms", QU =>, QD =>, CVU =>, CVD =>)
   END_RUNG
   RUNG wire#powerrail
      I_Contact( #EnTension )
   END_RUNG wire#w1
   // the same network as SCL:
   #TMP_EnTension(IN := #EnTension,   // "FB910_CNT_UHS"
                  R := NOT #EnTension,
                  PV := "V_TMP_EsperaEnTension",
                  BaseUnidades_ms := "CTE_BaseUnidades_1ms");
END_REGION

REGION Network 38: ERROR - Termico
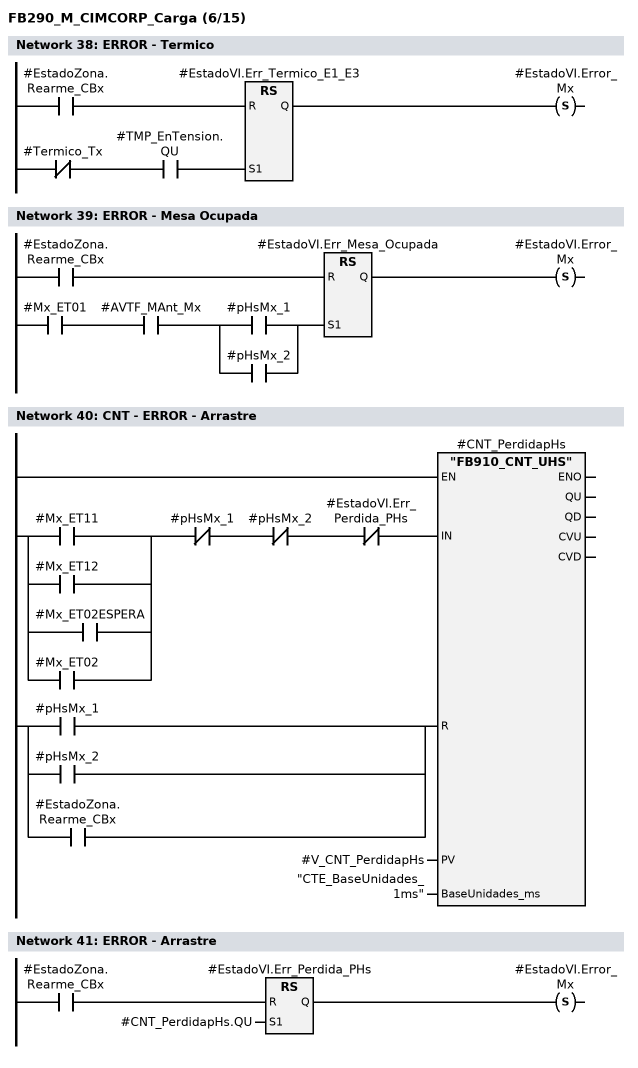
   RUNG wire#powerrail
      Contact( #EstadoZona.Rearme_CBx )
      S_RS(operand := #EstadoVI.Err_Termico_E1_E3, s1 := wire#w1)
      S_Coil( #EstadoVI.Error_Mx )
   END_RUNG
   RUNG wire#powerrail
      I_Contact( #Termico_Tx )
      Contact( #TMP_EnTension.QU )
   END_RUNG wire#w1
   // the same network as SCL:
   IF #EstadoZona.Rearme_CBx THEN
       #EstadoVI.Err_Termico_E1_E3 := FALSE;   // RS flip-flop
   END_IF;
   IF NOT #Termico_Tx AND #TMP_EnTension.QU THEN #EstadoVI.Err_Termico_E1_E3 := TRUE; END_IF;
   IF #EstadoVI.Err_Termico_E1_E3 THEN #EstadoVI.Error_Mx := TRUE; END_IF;
END_REGION

REGION Network 39: ERROR - Mesa Ocupada
   RUNG wire#powerrail
      Contact( #EstadoZona.Rearme_CBx )
      S_RS(operand := #EstadoVI.Err_Mesa_Ocupada, s1 := wire#w2)
      S_Coil( #EstadoVI.Error_Mx )
   END_RUNG
   RUNG wire#powerrail
      Contact( #Mx_ET01 )
      Contact( #AVTF_MAnt_Mx )
      wire#w1
      Contact( #pHsMx_1 )
   END_RUNG wire#w2
   RUNG wire#w1
      Contact( #pHsMx_2 )
   END_RUNG wire#w2
   // the same network as SCL:
   IF #EstadoZona.Rearme_CBx THEN
       #EstadoVI.Err_Mesa_Ocupada := FALSE;   // RS flip-flop
   END_IF;
   IF #Mx_ET01 AND #AVTF_MAnt_Mx AND (#pHsMx_1 OR #pHsMx_2) THEN #EstadoVI.Err_Mesa_Ocupada := TRUE; END_IF;
   IF #EstadoVI.Err_Mesa_Ocupada THEN #EstadoVI.Error_Mx := TRUE; END_IF;
END_REGION

REGION Network 40: CNT - ERROR - Arrastre
   RUNG wire#powerrail
      #CNT_PerdidapHs(IN := wire#w2, R := wire#w3, PV := #V_CNT_PerdidapHs, BaseUnidades_ms := "CTE_BaseUnidades_1ms", QU =>, QD =>, CVU =>, CVD =>)
   END_RUNG
   RUNG wire#powerrail
      Contact( #Mx_ET11 )
      wire#w1
      I_Contact( #pHsMx_1 )
      I_Contact( #pHsMx_2 )
      I_Contact( #EstadoVI.Err_Perdida_PHs )
   END_RUNG wire#w2
   RUNG wire#powerrail
      Contact( #Mx_ET12 )
   END_RUNG wire#w1
   RUNG wire#powerrail
      Contact( #Mx_ET02ESPERA )
   END_RUNG wire#w1
   RUNG wire#powerrail
      Contact( #Mx_ET02 )
   END_RUNG wire#w1
   RUNG wire#powerrail
      Contact( #pHsMx_1 )
   END_RUNG wire#w3
   RUNG wire#powerrail
      Contact( #pHsMx_2 )
   END_RUNG wire#w3
   RUNG wire#powerrail
      Contact( #EstadoZona.Rearme_CBx )
   END_RUNG wire#w3
   // the same network as SCL:
   #CNT_PerdidapHs(IN := (#Mx_ET11 OR #Mx_ET12 OR #Mx_ET02ESPERA OR #Mx_ET02) AND NOT #pHsMx_1 AND NOT #pHsMx_2 AND NOT #EstadoVI.Err_Perdida_PHs,   // "FB910_CNT_UHS"
                   R := #pHsMx_1 OR #pHsMx_2 OR #EstadoZona.Rearme_CBx,
                   PV := #V_CNT_PerdidapHs,
                   BaseUnidades_ms := "CTE_BaseUnidades_1ms");
END_REGION

REGION Network 41: ERROR - Arrastre
   RUNG wire#powerrail
      Contact( #EstadoZona.Rearme_CBx )
      S_RS(operand := #EstadoVI.Err_Perdida_PHs, s1 := #CNT_PerdidapHs.QU)
      S_Coil( #EstadoVI.Error_Mx )
   END_RUNG
   // the same network as SCL:
   IF #EstadoZona.Rearme_CBx THEN
       #EstadoVI.Err_Perdida_PHs := FALSE;   // RS flip-flop
   END_IF;
   IF #CNT_PerdidapHs.QU THEN #EstadoVI.Err_Perdida_PHs := TRUE; END_IF;
   IF #EstadoVI.Err_Perdida_PHs THEN #EstadoVI.Error_Mx := TRUE; END_IF;
END_REGION

REGION Network 42: TMP - ERROR - TimeOut Avance
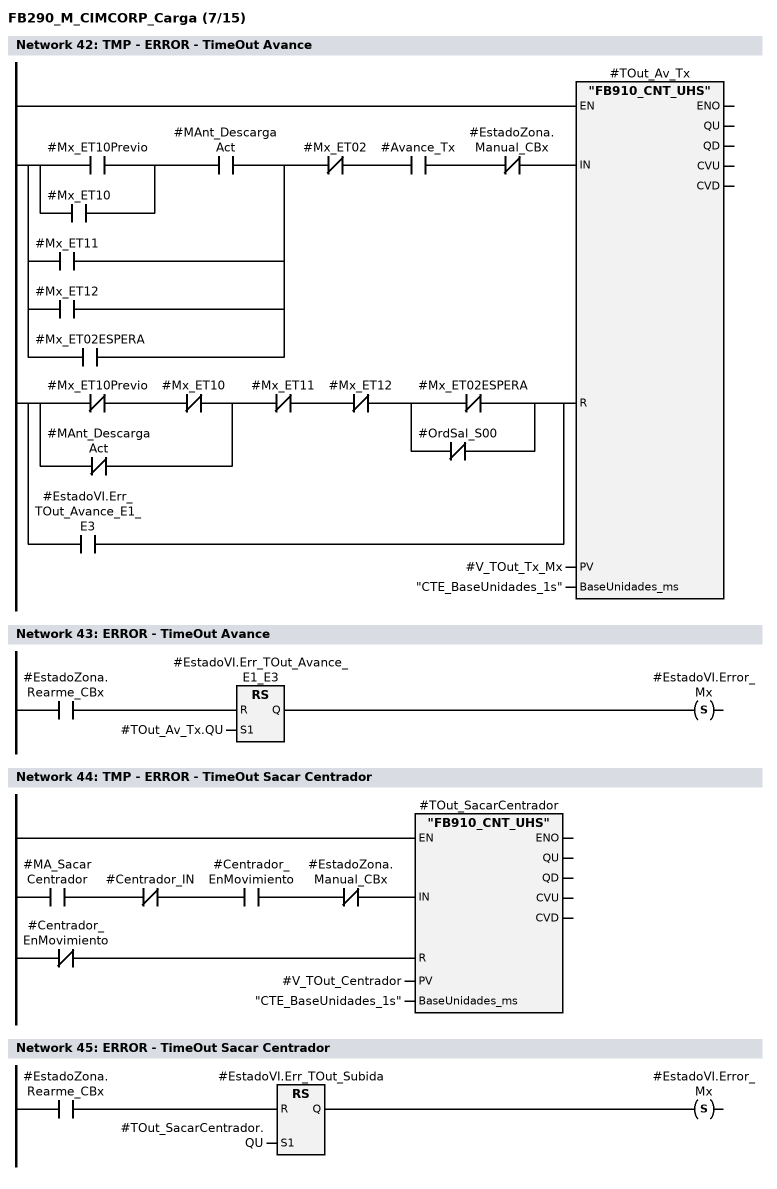
   RUNG wire#powerrail
      #TOut_Av_Tx(IN := wire#w3, R := wire#w6, PV := #V_TOut_Tx_Mx, BaseUnidades_ms := "CTE_BaseUnidades_1s", QU =>, QD =>, CVU =>, CVD =>)
   END_RUNG
   RUNG wire#powerrail
      Contact( #Mx_ET10Previo )
      wire#w1
      Contact( #MAnt_DescargaAct )
      wire#w2
      I_Contact( #Mx_ET02 )
      Contact( #Avance_Tx )
      I_Contact( #EstadoZona.Manual_CBx )
   END_RUNG wire#w3
   RUNG wire#powerrail
      Contact( #Mx_ET10 )
   END_RUNG wire#w1
   RUNG wire#powerrail
      Contact( #Mx_ET11 )
   END_RUNG wire#w2
   RUNG wire#powerrail
      Contact( #Mx_ET12 )
   END_RUNG wire#w2
   RUNG wire#powerrail
      Contact( #Mx_ET02ESPERA )
   END_RUNG wire#w2
   RUNG wire#powerrail
      I_Contact( #Mx_ET10Previo )
      I_Contact( #Mx_ET10 )
      wire#w4
      I_Contact( #Mx_ET11 )
      I_Contact( #Mx_ET12 )
      wire#w5
      I_Contact( #Mx_ET02ESPERA )
   END_RUNG wire#w6
   RUNG wire#powerrail
      I_Contact( #MAnt_DescargaAct )
   END_RUNG wire#w4
   RUNG wire#w5
      I_Contact( #OrdSal_S00 )
   END_RUNG wire#w6
   RUNG wire#powerrail
      Contact( #EstadoVI.Err_TOut_Avance_E1_E3 )
   END_RUNG wire#w6
   // the same network as SCL:
   #TOut_Av_Tx(IN := (((#Mx_ET10Previo OR #Mx_ET10) AND #MAnt_DescargaAct) OR #Mx_ET11 OR #Mx_ET12 OR #Mx_ET02ESPERA) AND NOT #Mx_ET02 AND #Avance_Tx AND NOT #EstadoZona.Manual_CBx,   // "FB910_CNT_UHS"
               R := (((NOT #Mx_ET10Previo AND NOT #Mx_ET10) OR NOT #MAnt_DescargaAct) AND NOT #Mx_ET11 AND NOT #Mx_ET12 AND (NOT #Mx_ET02ESPERA OR NOT #OrdSal_S00)) OR #EstadoVI.Err_TOut_Avance_E1_E3,
               PV := #V_TOut_Tx_Mx,
               BaseUnidades_ms := "CTE_BaseUnidades_1s");
END_REGION

REGION Network 43: ERROR - TimeOut Avance
   RUNG wire#powerrail
      Contact( #EstadoZona.Rearme_CBx )
      S_RS(operand := #EstadoVI.Err_TOut_Avance_E1_E3, s1 := #TOut_Av_Tx.QU)
      S_Coil( #EstadoVI.Error_Mx )
   END_RUNG
   // the same network as SCL:
   IF #EstadoZona.Rearme_CBx THEN
       #EstadoVI.Err_TOut_Avance_E1_E3 := FALSE;   // RS flip-flop
   END_IF;
   IF #TOut_Av_Tx.QU THEN #EstadoVI.Err_TOut_Avance_E1_E3 := TRUE; END_IF;
   IF #EstadoVI.Err_TOut_Avance_E1_E3 THEN #EstadoVI.Error_Mx := TRUE; END_IF;
END_REGION

REGION Network 44: TMP - ERROR - TimeOut Sacar Centrador
   RUNG wire#powerrail
      #TOut_SacarCentrador(IN := wire#w1, R := wire#w2, PV := #V_TOut_Centrador, BaseUnidades_ms := "CTE_BaseUnidades_1s", QU =>, QD =>, CVU =>, CVD =>)
   END_RUNG
   RUNG wire#powerrail
      Contact( #MA_SacarCentrador )
      I_Contact( #Centrador_IN )
      Contact( #Centrador_EnMovimiento )
      I_Contact( #EstadoZona.Manual_CBx )
   END_RUNG wire#w1
   RUNG wire#powerrail
      I_Contact( #Centrador_EnMovimiento )
   END_RUNG wire#w2
   // the same network as SCL:
   #TOut_SacarCentrador(IN := #MA_SacarCentrador AND NOT #Centrador_IN AND #Centrador_EnMovimiento AND NOT #EstadoZona.Manual_CBx,   // "FB910_CNT_UHS"
                        R := NOT #Centrador_EnMovimiento,
                        PV := #V_TOut_Centrador,
                        BaseUnidades_ms := "CTE_BaseUnidades_1s");
END_REGION

REGION Network 45: ERROR - TimeOut Sacar Centrador
   RUNG wire#powerrail
      Contact( #EstadoZona.Rearme_CBx )
      S_RS(operand := #EstadoVI.Err_TOut_Subida, s1 := #TOut_SacarCentrador.QU)
      S_Coil( #EstadoVI.Error_Mx )
   END_RUNG
   // the same network as SCL:
   IF #EstadoZona.Rearme_CBx THEN
       #EstadoVI.Err_TOut_Subida := FALSE;   // RS flip-flop
   END_IF;
   IF #TOut_SacarCentrador.QU THEN #EstadoVI.Err_TOut_Subida := TRUE; END_IF;
   IF #EstadoVI.Err_TOut_Subida THEN #EstadoVI.Error_Mx := TRUE; END_IF;
END_REGION

REGION Network 46: TMP - ERROR - TimeOut Recoger Centrador
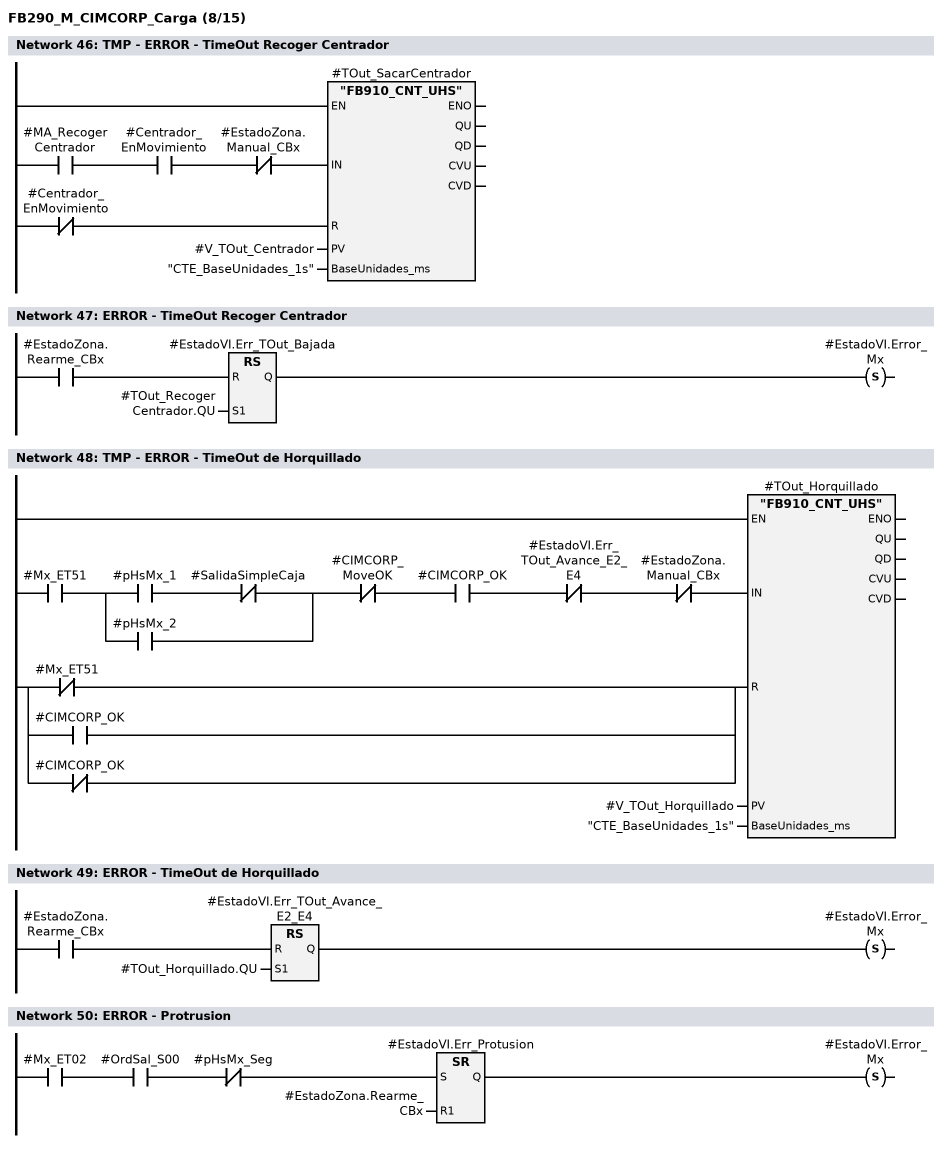
   RUNG wire#powerrail
      #TOut_SacarCentrador(IN := wire#w1, R := wire#w2, PV := #V_TOut_Centrador, BaseUnidades_ms := "CTE_BaseUnidades_1s", QU =>, QD =>, CVU =>, CVD =>)
   END_RUNG
   RUNG wire#powerrail
      Contact( #MA_RecogerCentrador )
      Contact( #Centrador_EnMovimiento )
      I_Contact( #EstadoZona.Manual_CBx )
   END_RUNG wire#w1
   RUNG wire#powerrail
      I_Contact( #Centrador_EnMovimiento )
   END_RUNG wire#w2
   // the same network as SCL:
   #TOut_SacarCentrador(IN := #MA_RecogerCentrador AND #Centrador_EnMovimiento AND NOT #EstadoZona.Manual_CBx,   // "FB910_CNT_UHS"
                        R := NOT #Centrador_EnMovimiento,
                        PV := #V_TOut_Centrador,
                        BaseUnidades_ms := "CTE_BaseUnidades_1s");
END_REGION

REGION Network 47: ERROR - TimeOut Recoger Centrador
   RUNG wire#powerrail
      Contact( #EstadoZona.Rearme_CBx )
      S_RS(operand := #EstadoVI.Err_TOut_Bajada, s1 := #TOut_RecogerCentrador.QU)
      S_Coil( #EstadoVI.Error_Mx )
   END_RUNG
   // the same network as SCL:
   IF #EstadoZona.Rearme_CBx THEN
       #EstadoVI.Err_TOut_Bajada := FALSE;   // RS flip-flop
   END_IF;
   IF #TOut_RecogerCentrador.QU THEN #EstadoVI.Err_TOut_Bajada := TRUE; END_IF;
   IF #EstadoVI.Err_TOut_Bajada THEN #EstadoVI.Error_Mx := TRUE; END_IF;
END_REGION

REGION Network 48: TMP - ERROR - TimeOut de Horquillado
   RUNG wire#powerrail
      #TOut_Horquillado(IN := wire#w3, R := wire#w4, PV := #V_TOut_Horquillado, BaseUnidades_ms := "CTE_BaseUnidades_1s", QU =>, QD =>, CVU =>, CVD =>)
   END_RUNG
   RUNG wire#powerrail
      Contact( #Mx_ET51 )
      wire#w1
      Contact( #pHsMx_1 )
      I_Contact( #SalidaSimpleCaja )
      wire#w2
      I_Contact( #CIMCORP_MoveOK )
      Contact( #CIMCORP_OK )
      I_Contact( #EstadoVI.Err_TOut_Avance_E2_E4 )
      I_Contact( #EstadoZona.Manual_CBx )
   END_RUNG wire#w3
   RUNG wire#w1
      Contact( #pHsMx_2 )
   END_RUNG wire#w2
   RUNG wire#powerrail
      I_Contact( #Mx_ET51 )
   END_RUNG wire#w4
   RUNG wire#powerrail
      Contact( #CIMCORP_OK )
   END_RUNG wire#w4
   RUNG wire#powerrail
      I_Contact( #CIMCORP_OK )
   END_RUNG wire#w4
   // the same network as SCL:
   #TOut_Horquillado(IN := #Mx_ET51 AND ((#pHsMx_1 AND NOT #SalidaSimpleCaja) OR #pHsMx_2) AND NOT #CIMCORP_MoveOK AND #CIMCORP_OK AND NOT #EstadoVI.Err_TOut_Avance_E2_E4 AND NOT #EstadoZona.Manual_CBx,   // "FB910_CNT_UHS"
                     R := NOT #Mx_ET51 OR #CIMCORP_OK OR NOT #CIMCORP_OK,
                     PV := #V_TOut_Horquillado,
                     BaseUnidades_ms := "CTE_BaseUnidades_1s");
END_REGION

REGION Network 49: ERROR - TimeOut de Horquillado
   RUNG wire#powerrail
      Contact( #EstadoZona.Rearme_CBx )
      S_RS(operand := #EstadoVI.Err_TOut_Avance_E2_E4, s1 := #TOut_Horquillado.QU)
      S_Coil( #EstadoVI.Error_Mx )
   END_RUNG
   // the same network as SCL:
   IF #EstadoZona.Rearme_CBx THEN
       #EstadoVI.Err_TOut_Avance_E2_E4 := FALSE;   // RS flip-flop
   END_IF;
   IF #TOut_Horquillado.QU THEN #EstadoVI.Err_TOut_Avance_E2_E4 := TRUE; END_IF;
   IF #EstadoVI.Err_TOut_Avance_E2_E4 THEN #EstadoVI.Error_Mx := TRUE; END_IF;
END_REGION

REGION Network 50: ERROR - Protrusion
   RUNG wire#powerrail
      Contact( #Mx_ET02 )
      Contact( #OrdSal_S00 )
      I_Contact( #pHsMx_Seg )
      S_SR(operand := #EstadoVI.Err_Protusion, r1 := #EstadoZona.Rearme_CBx)
      S_Coil( #EstadoVI.Error_Mx )
   END_RUNG
   // the same network as SCL:
   IF #Mx_ET02 AND #OrdSal_S00 AND NOT #pHsMx_Seg THEN
       #EstadoVI.Err_Protusion := TRUE;   // SR flip-flop
   END_IF;
   IF #EstadoZona.Rearme_CBx THEN #EstadoVI.Err_Protusion := FALSE; END_IF;
   IF #EstadoVI.Err_Protusion THEN #EstadoVI.Error_Mx := TRUE; END_IF;
END_REGION

REGION Network 51: CONTADOR DE SEGURIDAD DE PRESENCIA - CNTSeg_pHsMx
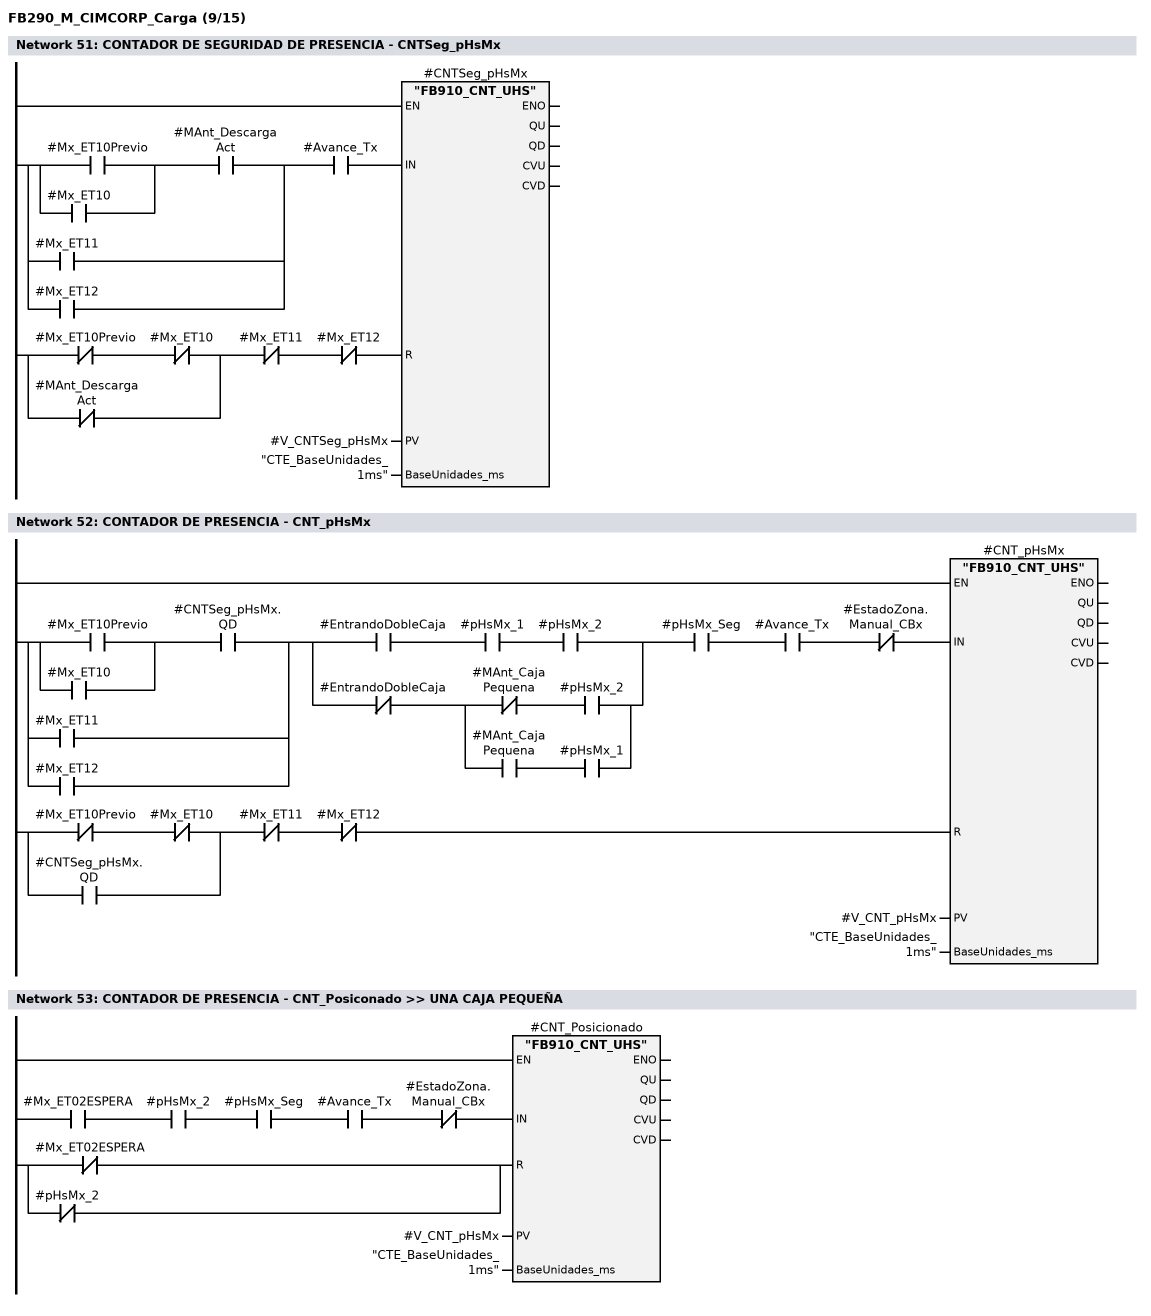
   RUNG wire#powerrail
      #CNTSeg_pHsMx(IN := wire#w3, R := wire#w5, PV := #V_CNTSeg_pHsMx, BaseUnidades_ms := "CTE_BaseUnidades_1ms", QU =>, QD =>, CVU =>, CVD =>)
   END_RUNG
   RUNG wire#powerrail
      Contact( #Mx_ET10Previo )
      wire#w1
      Contact( #MAnt_DescargaAct )
      wire#w2
      Contact( #Avance_Tx )
   END_RUNG wire#w3
   RUNG wire#powerrail
      Contact( #Mx_ET10 )
   END_RUNG wire#w1
   RUNG wire#powerrail
      Contact( #Mx_ET11 )
   END_RUNG wire#w2
   RUNG wire#powerrail
      Contact( #Mx_ET12 )
   END_RUNG wire#w2
   RUNG wire#powerrail
      I_Contact( #Mx_ET10Previo )
      I_Contact( #Mx_ET10 )
      wire#w4
      I_Contact( #Mx_ET11 )
      I_Contact( #Mx_ET12 )
   END_RUNG wire#w5
   RUNG wire#powerrail
      I_Contact( #MAnt_DescargaAct )
   END_RUNG wire#w4
   // the same network as SCL:
   #CNTSeg_pHsMx(IN := (((#Mx_ET10Previo OR #Mx_ET10) AND #MAnt_DescargaAct) OR #Mx_ET11 OR #Mx_ET12) AND #Avance_Tx,   // "FB910_CNT_UHS"
                 R := ((NOT #Mx_ET10Previo AND NOT #Mx_ET10) OR NOT #MAnt_DescargaAct) AND NOT #Mx_ET11 AND NOT #Mx_ET12,
                 PV := #V_CNTSeg_pHsMx,
                 BaseUnidades_ms := "CTE_BaseUnidades_1ms");
END_REGION

REGION Network 52: CONTADOR DE PRESENCIA - CNT_pHsMx
   RUNG wire#powerrail
      #CNT_pHsMx(IN := wire#w5, R := wire#w7, PV := #V_CNT_pHsMx, BaseUnidades_ms := "CTE_BaseUnidades_1ms", QU =>, QD =>, CVU =>, CVD =>)
   END_RUNG
   RUNG wire#powerrail
      Contact( #Mx_ET10Previo )
      wire#w1
      Contact( #CNTSeg_pHsMx.QD )
      wire#w2
      Contact( #EntrandoDobleCaja )
      Contact( #pHsMx_1 )
      Contact( #pHsMx_2 )
      wire#w3
      Contact( #pHsMx_Seg )
      Contact( #Avance_Tx )
      I_Contact( #EstadoZona.Manual_CBx )
   END_RUNG wire#w5
   RUNG wire#powerrail
      Contact( #Mx_ET10 )
   END_RUNG wire#w1
   RUNG wire#powerrail
      Contact( #Mx_ET11 )
   END_RUNG wire#w2
   RUNG wire#powerrail
      Contact( #Mx_ET12 )
   END_RUNG wire#w2
   RUNG wire#w2
      I_Contact( #EntrandoDobleCaja )
      wire#w4
      I_Contact( #MAnt_CajaPequena )
      Contact( #pHsMx_2 )
   END_RUNG wire#w3
   RUNG wire#w4
      Contact( #MAnt_CajaPequena )
      Contact( #pHsMx_1 )
   END_RUNG wire#w3
   RUNG wire#powerrail
      I_Contact( #Mx_ET10Previo )
      I_Contact( #Mx_ET10 )
      wire#w6
      I_Contact( #Mx_ET11 )
      I_Contact( #Mx_ET12 )
   END_RUNG wire#w7
   RUNG wire#powerrail
      Contact( #CNTSeg_pHsMx.QD )
   END_RUNG wire#w6
   // the same network as SCL:
   #CNT_pHsMx(IN := (((#Mx_ET10Previo OR #Mx_ET10) AND #CNTSeg_pHsMx.QD) OR #Mx_ET11 OR #Mx_ET12) AND ((#EntrandoDobleCaja AND #pHsMx_1 AND #pHsMx_2) OR (NOT #EntrandoDobleCaja AND ((NOT #MAnt_CajaPequena AND #pHsMx_2) OR (#MAnt_CajaPequena AND #pHsMx_1)))) AND #pHsMx_Seg AND #Avance_Tx AND NOT #EstadoZona.Manual_CBx,   // "FB910_CNT_UHS"
              R := ((NOT #Mx_ET10Previo AND NOT #Mx_ET10) OR #CNTSeg_pHsMx.QD) AND NOT #Mx_ET11 AND NOT #Mx_ET12,
              PV := #V_CNT_pHsMx,
              BaseUnidades_ms := "CTE_BaseUnidades_1ms");
END_REGION

REGION Network 53: CONTADOR DE PRESENCIA - CNT_Posiconado >> UNA CAJA PEQUEÑA
   RUNG wire#powerrail
      #CNT_Posicionado(IN := wire#w1, R := wire#w2, PV := #V_CNT_pHsMx, BaseUnidades_ms := "CTE_BaseUnidades_1ms", QU =>, QD =>, CVU =>, CVD =>)
   END_RUNG
   RUNG wire#powerrail
      Contact( #Mx_ET02ESPERA )
      Contact( #pHsMx_2 )
      Contact( #pHsMx_Seg )
      Contact( #Avance_Tx )
      I_Contact( #EstadoZona.Manual_CBx )
   END_RUNG wire#w1
   RUNG wire#powerrail
      I_Contact( #Mx_ET02ESPERA )
   END_RUNG wire#w2
   RUNG wire#powerrail
      I_Contact( #pHsMx_2 )
   END_RUNG wire#w2
   // the same network as SCL:
   #CNT_Posicionado(IN := #Mx_ET02ESPERA AND #pHsMx_2 AND #pHsMx_Seg AND #Avance_Tx AND NOT #EstadoZona.Manual_CBx,   // "FB910_CNT_UHS"
                    R := NOT #Mx_ET02ESPERA OR NOT #pHsMx_2,
                    PV := #V_CNT_pHsMx,
                    BaseUnidades_ms := "CTE_BaseUnidades_1ms");
END_REGION

REGION Network 54: CONTROL DEL COMPACTADO - Memoria de Centrador IN >> PREPARADO PARA EL COMPACTADO
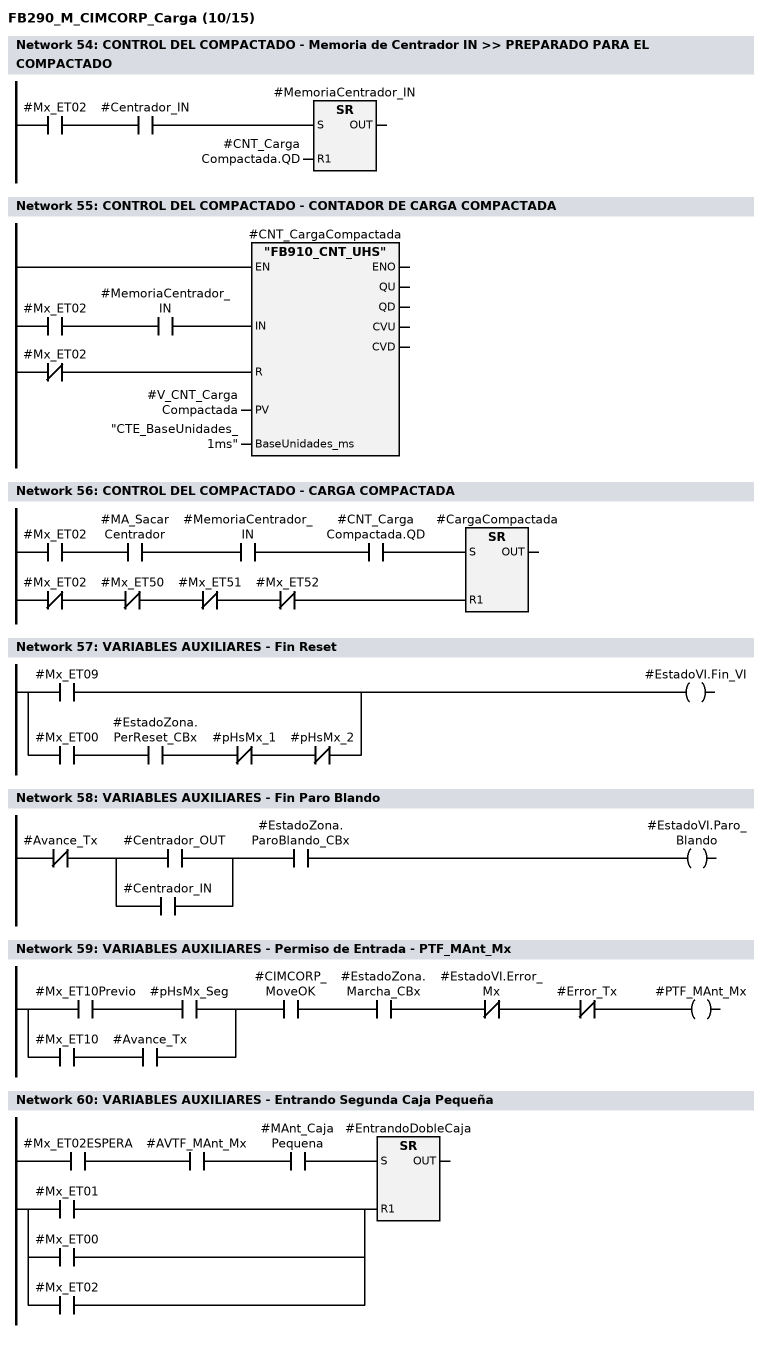
   RUNG wire#powerrail
      Contact( #Mx_ET02 )
      Contact( #Centrador_IN )
      S_SR(operand := #MemoriaCentrador_IN, r1 := #CNT_CargaCompactada.QD)
   END_RUNG
   // the same network as SCL:
   IF #Mx_ET02 AND #Centrador_IN THEN
       #MemoriaCentrador_IN := TRUE;   // SR flip-flop
   END_IF;
   IF #CNT_CargaCompactada.QD THEN #MemoriaCentrador_IN := FALSE; END_IF;
END_REGION

REGION Network 55: CONTROL DEL COMPACTADO - CONTADOR DE CARGA COMPACTADA
   RUNG wire#powerrail
      #CNT_CargaCompactada(IN := wire#w1, R := wire#w2, PV := #V_CNT_CargaCompactada, BaseUnidades_ms := "CTE_BaseUnidades_1ms", QU =>, QD =>, CVU =>, CVD =>)
   END_RUNG
   RUNG wire#powerrail
      Contact( #Mx_ET02 )
      Contact( #MemoriaCentrador_IN )
   END_RUNG wire#w1
   RUNG wire#powerrail
      I_Contact( #Mx_ET02 )
   END_RUNG wire#w2
   // the same network as SCL:
   #CNT_CargaCompactada(IN := #Mx_ET02 AND #MemoriaCentrador_IN,   // "FB910_CNT_UHS"
                        R := NOT #Mx_ET02,
                        PV := #V_CNT_CargaCompactada,
                        BaseUnidades_ms := "CTE_BaseUnidades_1ms");
END_REGION

REGION Network 56: CONTROL DEL COMPACTADO - CARGA COMPACTADA
   RUNG wire#powerrail
      Contact( #Mx_ET02 )
      Contact( #MA_SacarCentrador )
      Contact( #MemoriaCentrador_IN )
      Contact( #CNT_CargaCompactada.QD )
      S_SR(operand := #CargaCompactada, r1 := wire#w1)
   END_RUNG
   RUNG wire#powerrail
      I_Contact( #Mx_ET02 )
      I_Contact( #Mx_ET50 )
      I_Contact( #Mx_ET51 )
      I_Contact( #Mx_ET52 )
   END_RUNG wire#w1
   // the same network as SCL:
   IF #Mx_ET02 AND #MA_SacarCentrador AND #MemoriaCentrador_IN AND #CNT_CargaCompactada.QD THEN
       #CargaCompactada := TRUE;   // SR flip-flop
   END_IF;
   IF NOT #Mx_ET02 AND NOT #Mx_ET50 AND NOT #Mx_ET51 AND NOT #Mx_ET52 THEN #CargaCompactada := FALSE; END_IF;
END_REGION

REGION Network 57: VARIABLES AUXILIARES - Fin Reset
   RUNG wire#powerrail
      Contact( #Mx_ET09 )
      wire#w1
      Coil( #EstadoVI.Fin_VI )
   END_RUNG
   RUNG wire#powerrail
      Contact( #Mx_ET00 )
      Contact( #EstadoZona.PerReset_CBx )
      I_Contact( #pHsMx_1 )
      I_Contact( #pHsMx_2 )
   END_RUNG wire#w1
   // the same network as SCL:
   #EstadoVI.Fin_VI := #Mx_ET09 OR (#Mx_ET00 AND #EstadoZona.PerReset_CBx AND NOT #pHsMx_1 AND NOT #pHsMx_2);
END_REGION

REGION Network 58: VARIABLES AUXILIARES - Fin Paro Blando
   RUNG wire#powerrail
      I_Contact( #Avance_Tx )
      wire#w1
      Contact( #Centrador_OUT )
      wire#w2
      Contact( #EstadoZona.ParoBlando_CBx )
      Coil( #EstadoVI.Paro_Blando )
   END_RUNG
   RUNG wire#w1
      Contact( #Centrador_IN )
   END_RUNG wire#w2
   // the same network as SCL:
   #EstadoVI.Paro_Blando := NOT #Avance_Tx AND (#Centrador_OUT OR #Centrador_IN) AND #EstadoZona.ParoBlando_CBx;
END_REGION

REGION Network 59: VARIABLES AUXILIARES - Permiso de Entrada - PTF_MAnt_Mx
   RUNG wire#powerrail
      Contact( #Mx_ET10Previo )
      Contact( #pHsMx_Seg )
      wire#w1
      Contact( #CIMCORP_MoveOK )
      Contact( #EstadoZona.Marcha_CBx )
      I_Contact( #EstadoVI.Error_Mx )
      I_Contact( #Error_Tx )
      Coil( #PTF_MAnt_Mx )
   END_RUNG
   RUNG wire#powerrail
      Contact( #Mx_ET10 )
      Contact( #Avance_Tx )
   END_RUNG wire#w1
   // the same network as SCL:
   #PTF_MAnt_Mx := ((#Mx_ET10Previo AND #pHsMx_Seg) OR (#Mx_ET10 AND #Avance_Tx)) AND #CIMCORP_MoveOK AND #EstadoZona.Marcha_CBx AND NOT #EstadoVI.Error_Mx AND NOT #Error_Tx;
END_REGION

REGION Network 60: VARIABLES AUXILIARES - Entrando Segunda Caja Pequeña
   RUNG wire#powerrail
      Contact( #Mx_ET02ESPERA )
      Contact( #AVTF_MAnt_Mx )
      Contact( #MAnt_CajaPequena )
      S_SR(operand := #EntrandoDobleCaja, r1 := wire#w1)
   END_RUNG
   RUNG wire#powerrail
      Contact( #Mx_ET01 )
   END_RUNG wire#w1
   RUNG wire#powerrail
      Contact( #Mx_ET00 )
   END_RUNG wire#w1
   RUNG wire#powerrail
      Contact( #Mx_ET02 )
   END_RUNG wire#w1
   // the same network as SCL:
   IF #Mx_ET02ESPERA AND #AVTF_MAnt_Mx AND #MAnt_CajaPequena THEN
       #EntrandoDobleCaja := TRUE;   // SR flip-flop
   END_IF;
   IF #Mx_ET01 OR #Mx_ET00 OR #Mx_ET02 THEN #EntrandoDobleCaja := FALSE; END_IF;
END_REGION

REGION Network 61: VARIABLES AUXILIARES - Salida de Caja Grande
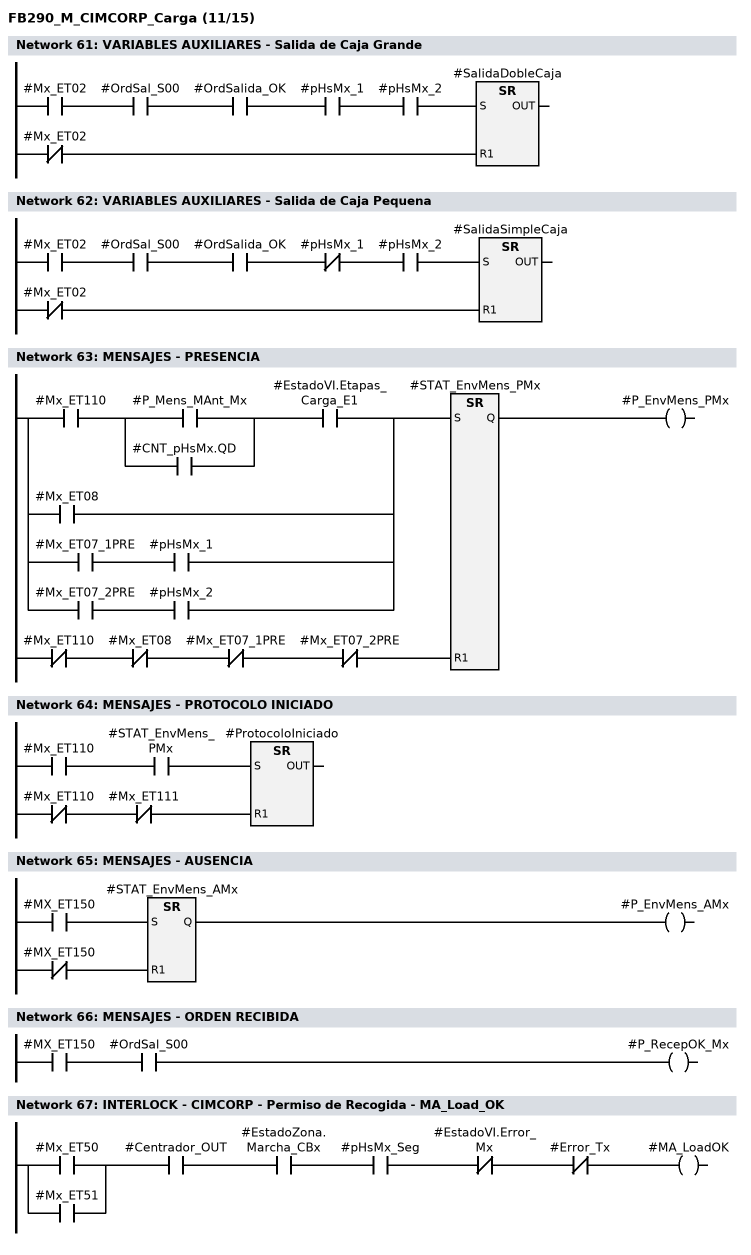
   RUNG wire#powerrail
      Contact( #Mx_ET02 )
      Contact( #OrdSal_S00 )
      Contact( #OrdSalida_OK )
      Contact( #pHsMx_1 )
      Contact( #pHsMx_2 )
      S_SR(operand := #SalidaDobleCaja, r1 := wire#w1)
   END_RUNG
   RUNG wire#powerrail
      I_Contact( #Mx_ET02 )
   END_RUNG wire#w1
   // the same network as SCL:
   IF #Mx_ET02 AND #OrdSal_S00 AND #OrdSalida_OK AND #pHsMx_1 AND #pHsMx_2 THEN
       #SalidaDobleCaja := TRUE;   // SR flip-flop
   END_IF;
   IF NOT #Mx_ET02 THEN #SalidaDobleCaja := FALSE; END_IF;
END_REGION

REGION Network 62: VARIABLES AUXILIARES - Salida de Caja Pequena
   RUNG wire#powerrail
      Contact( #Mx_ET02 )
      Contact( #OrdSal_S00 )
      Contact( #OrdSalida_OK )
      I_Contact( #pHsMx_1 )
      Contact( #pHsMx_2 )
      S_SR(operand := #SalidaSimpleCaja, r1 := wire#w1)
   END_RUNG
   RUNG wire#powerrail
      I_Contact( #Mx_ET02 )
   END_RUNG wire#w1
   // the same network as SCL:
   IF #Mx_ET02 AND #OrdSal_S00 AND #OrdSalida_OK AND NOT #pHsMx_1 AND #pHsMx_2 THEN
       #SalidaSimpleCaja := TRUE;   // SR flip-flop
   END_IF;
   IF NOT #Mx_ET02 THEN #SalidaSimpleCaja := FALSE; END_IF;
END_REGION

REGION Network 63: MENSAJES - PRESENCIA
   RUNG wire#powerrail
      Contact( #Mx_ET110 )
      wire#w1
      Contact( #P_Mens_MAnt_Mx )
      wire#w2
      Contact( #EstadoVI.Etapas_Carga_E1 )
      wire#w3
      S_SR(operand := #STAT_EnvMens_PMx, r1 := wire#w4)
      Coil( #P_EnvMens_PMx )
   END_RUNG
   RUNG wire#w1
      Contact( #CNT_pHsMx.QD )
   END_RUNG wire#w2
   RUNG wire#powerrail
      Contact( #Mx_ET08 )
   END_RUNG wire#w3
   RUNG wire#powerrail
      Contact( #Mx_ET07_1PRE )
      Contact( #pHsMx_1 )
   END_RUNG wire#w3
   RUNG wire#powerrail
      Contact( #Mx_ET07_2PRE )
      Contact( #pHsMx_2 )
   END_RUNG wire#w3
   RUNG wire#powerrail
      I_Contact( #Mx_ET110 )
      I_Contact( #Mx_ET08 )
      I_Contact( #Mx_ET07_1PRE )
      I_Contact( #Mx_ET07_2PRE )
   END_RUNG wire#w4
   // the same network as SCL:
   IF (#Mx_ET110 AND (#P_Mens_MAnt_Mx OR #CNT_pHsMx.QD) AND #EstadoVI.Etapas_Carga_E1) OR #Mx_ET08 OR (#Mx_ET07_1PRE AND #pHsMx_1) OR (#Mx_ET07_2PRE AND #pHsMx_2) THEN
       #STAT_EnvMens_PMx := TRUE;   // SR flip-flop
   END_IF;
   IF NOT #Mx_ET110 AND NOT #Mx_ET08 AND NOT #Mx_ET07_1PRE AND NOT #Mx_ET07_2PRE THEN
       #STAT_EnvMens_PMx := FALSE;
   END_IF;
   #P_EnvMens_PMx := #STAT_EnvMens_PMx;
END_REGION

REGION Network 64: MENSAJES - PROTOCOLO INICIADO
   RUNG wire#powerrail
      Contact( #Mx_ET110 )
      Contact( #STAT_EnvMens_PMx )
      S_SR(operand := #ProtocoloIniciado, r1 := wire#w1)
   END_RUNG
   RUNG wire#powerrail
      I_Contact( #Mx_ET110 )
      I_Contact( #Mx_ET111 )
   END_RUNG wire#w1
   // the same network as SCL:
   IF #Mx_ET110 AND #STAT_EnvMens_PMx THEN
       #ProtocoloIniciado := TRUE;   // SR flip-flop
   END_IF;
   IF NOT #Mx_ET110 AND NOT #Mx_ET111 THEN #ProtocoloIniciado := FALSE; END_IF;
END_REGION

REGION Network 65: MENSAJES - AUSENCIA
   RUNG wire#powerrail
      Contact( #MX_ET150 )
      S_SR(operand := #STAT_EnvMens_AMx, r1 := wire#w1)
      Coil( #P_EnvMens_AMx )
   END_RUNG
   RUNG wire#powerrail
      I_Contact( #MX_ET150 )
   END_RUNG wire#w1
   // the same network as SCL:
   IF #MX_ET150 THEN
       #STAT_EnvMens_AMx := TRUE;   // SR flip-flop
   END_IF;
   IF NOT #MX_ET150 THEN #STAT_EnvMens_AMx := FALSE; END_IF;
   #P_EnvMens_AMx := #STAT_EnvMens_AMx;
END_REGION

REGION Network 66: MENSAJES - ORDEN RECIBIDA
   RUNG wire#powerrail
      Contact( #MX_ET150 )
      Contact( #OrdSal_S00 )
      Coil( #P_RecepOK_Mx )
   END_RUNG
   // the same network as SCL:
   #P_RecepOK_Mx := #MX_ET150 AND #OrdSal_S00;
END_REGION

REGION Network 67: INTERLOCK - CIMCORP - Permiso de Recogida - MA_Load_OK
   RUNG wire#powerrail
      Contact( #Mx_ET50 )
      wire#w1
      Contact( #Centrador_OUT )
      Contact( #EstadoZona.Marcha_CBx )
      Contact( #pHsMx_Seg )
      I_Contact( #EstadoVI.Error_Mx )
      I_Contact( #Error_Tx )
      Coil( #MA_LoadOK )
   END_RUNG
   RUNG wire#powerrail
      Contact( #Mx_ET51 )
   END_RUNG wire#w1
   // the same network as SCL:
   #MA_LoadOK := (#Mx_ET50 OR #Mx_ET51) AND #Centrador_OUT AND #EstadoZona.Marcha_CBx AND #pHsMx_Seg AND NOT #EstadoVI.Error_Mx AND NOT #Error_Tx;
END_REGION

REGION Network 68: SALIDAS - Avance Tx
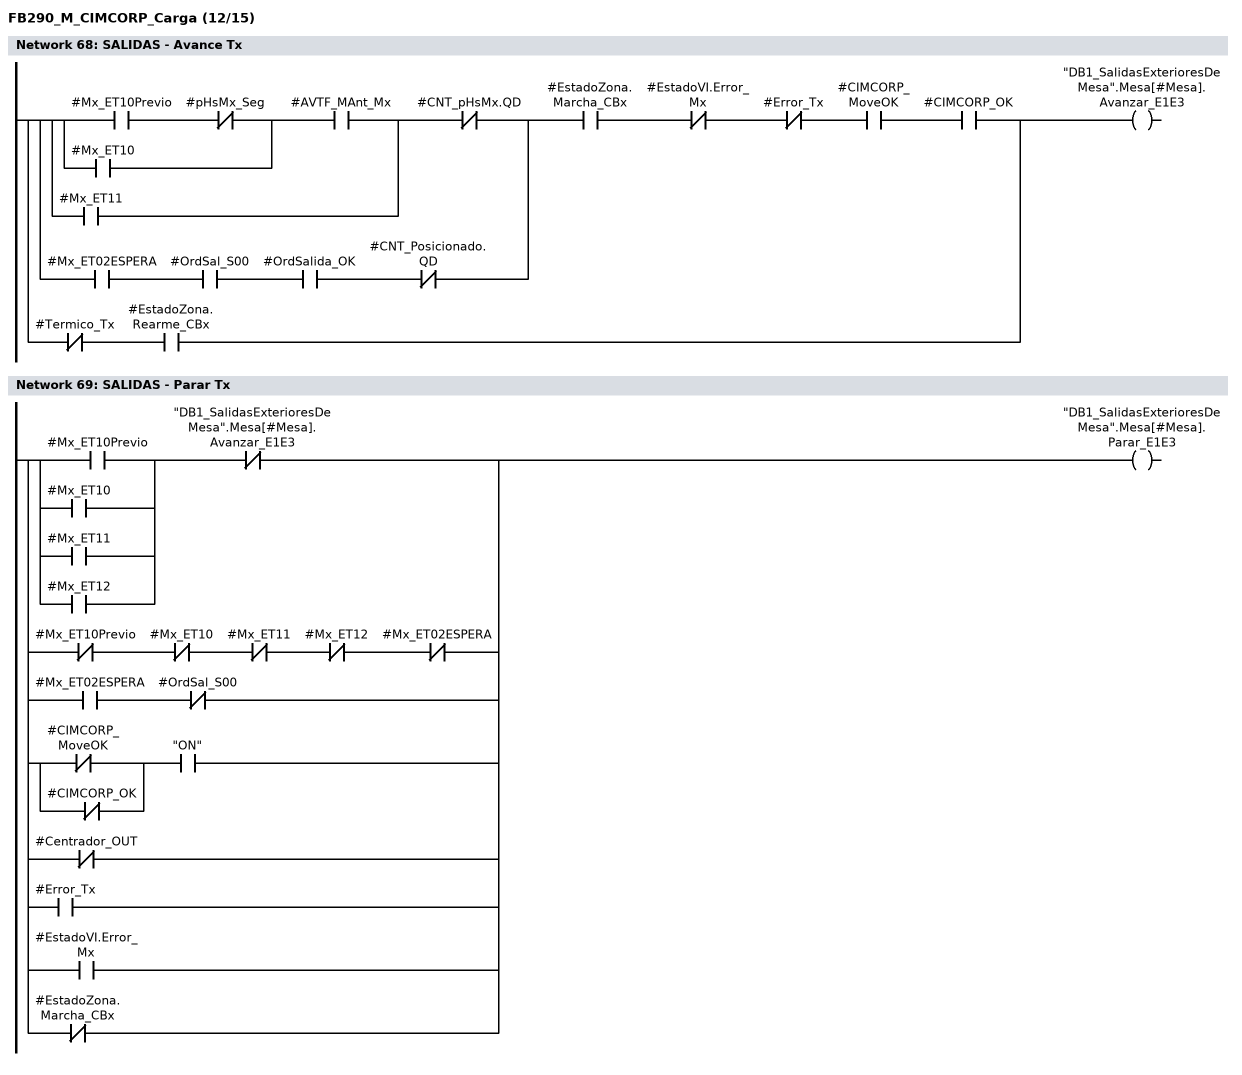
   RUNG wire#powerrail
      Contact( #Mx_ET10Previo )
      I_Contact( #pHsMx_Seg )
      wire#w1
      Contact( #AVTF_MAnt_Mx )
      wire#w2
      I_Contact( #CNT_pHsMx.QD )
      wire#w3
      Contact( #EstadoZona.Marcha_CBx )
      I_Contact( #EstadoVI.Error_Mx )
      I_Contact( #Error_Tx )
      Contact( #CIMCORP_MoveOK )
      Contact( #CIMCORP_OK )
      wire#w4
      Coil( "DB1_SalidasExterioresDeMesa".Mesa[#Mesa].Avanzar_E1E3 )
   END_RUNG
   RUNG wire#powerrail
      Contact( #Mx_ET10 )
   END_RUNG wire#w1
   RUNG wire#powerrail
      Contact( #Mx_ET11 )
   END_RUNG wire#w2
   RUNG wire#powerrail
      Contact( #Mx_ET02ESPERA )
      Contact( #OrdSal_S00 )
      Contact( #OrdSalida_OK )
      I_Contact( #CNT_Posicionado.QD )
   END_RUNG wire#w3
   RUNG wire#powerrail
      I_Contact( #Termico_Tx )
      Contact( #EstadoZona.Rearme_CBx )
   END_RUNG wire#w4
   // the same network as SCL:
   "DB1_SalidasExterioresDeMesa".Mesa[#Mesa].Avanzar_E1E3 := (((((((#Mx_ET10Previo AND NOT #pHsMx_Seg) OR #Mx_ET10) AND #AVTF_MAnt_Mx) OR #Mx_ET11) AND NOT #CNT_pHsMx.QD) OR (#Mx_ET02ESPERA AND #OrdSal_S00 AND #OrdSalida_OK AND NOT #CNT_Posicionado.QD)) AND #EstadoZona.Marcha_CBx AND NOT #EstadoVI.Error_Mx AND NOT #Error_Tx AND #CIMCORP_MoveOK AND #CIMCORP_OK) OR (NOT #Termico_Tx AND #EstadoZona.Rearme_CBx);
END_REGION

REGION Network 69: SALIDAS - Parar Tx
   RUNG wire#powerrail
      Contact( #Mx_ET10Previo )
      wire#w1
      I_Contact( "DB1_SalidasExterioresDeMesa".Mesa[#Mesa].Avanzar_E1E3 )
      wire#w2
      Coil( "DB1_SalidasExterioresDeMesa".Mesa[#Mesa].Parar_E1E3 )
   END_RUNG
   RUNG wire#powerrail
      Contact( #Mx_ET10 )
   END_RUNG wire#w1
   RUNG wire#powerrail
      Contact( #Mx_ET11 )
   END_RUNG wire#w1
   RUNG wire#powerrail
      Contact( #Mx_ET12 )
   END_RUNG wire#w1
   RUNG wire#powerrail
      I_Contact( #Mx_ET10Previo )
      I_Contact( #Mx_ET10 )
      I_Contact( #Mx_ET11 )
      I_Contact( #Mx_ET12 )
      I_Contact( #Mx_ET02ESPERA )
   END_RUNG wire#w2
   RUNG wire#powerrail
      Contact( #Mx_ET02ESPERA )
      I_Contact( #OrdSal_S00 )
   END_RUNG wire#w2
   RUNG wire#powerrail
      I_Contact( #CIMCORP_MoveOK )
      wire#w3
      Contact( "ON" )
   END_RUNG wire#w2
   RUNG wire#powerrail
      I_Contact( #CIMCORP_OK )
   END_RUNG wire#w3
   RUNG wire#powerrail
      I_Contact( #Centrador_OUT )
   END_RUNG wire#w2
   RUNG wire#powerrail
      Contact( #Error_Tx )
   END_RUNG wire#w2
   RUNG wire#powerrail
      Contact( #EstadoVI.Error_Mx )
   END_RUNG wire#w2
   RUNG wire#powerrail
      I_Contact( #EstadoZona.Marcha_CBx )
   END_RUNG wire#w2
   // the same network as SCL:
   "DB1_SalidasExterioresDeMesa".Mesa[#Mesa].Parar_E1E3 := ((#Mx_ET10Previo OR #Mx_ET10 OR #Mx_ET11 OR #Mx_ET12) AND NOT "DB1_SalidasExterioresDeMesa".Mesa[#Mesa].Avanzar_E1E3) OR (NOT #Mx_ET10Previo AND NOT #Mx_ET10 AND NOT #Mx_ET11 AND NOT #Mx_ET12 AND NOT #Mx_ET02ESPERA) OR (#Mx_ET02ESPERA AND NOT #OrdSal_S00) OR ((NOT #CIMCORP_MoveOK OR NOT #CIMCORP_OK) AND "ON") OR NOT #Centrador_OUT OR #Error_Tx OR #EstadoVI.Error_Mx OR NOT #EstadoZona.Marcha_CBx;
END_REGION

REGION Network 70: SALIDAS - Valor Frecuencia Lenta E1E3
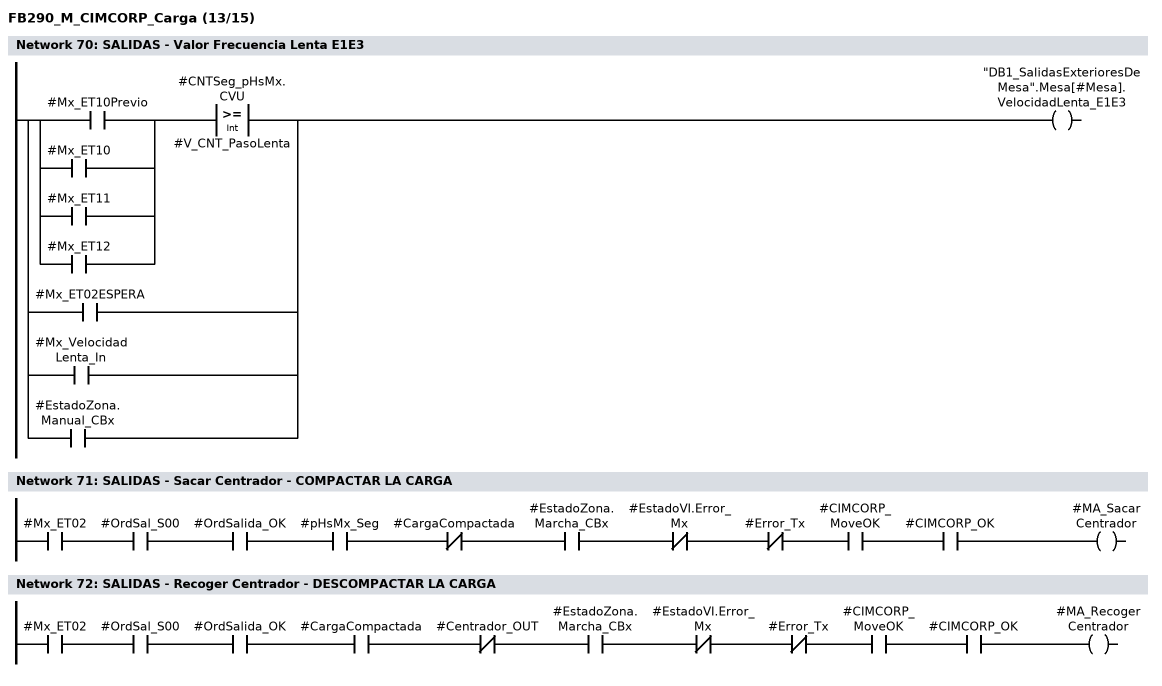
   RUNG wire#powerrail
      Contact( #Mx_ET10Previo )
      wire#w1
      { S7_Templates := "SrcType := Int" } GE_Contact(in1 := #CNTSeg_pHsMx.CVU, in2 := #V_CNT_PasoLenta)
      wire#w2
      Coil( "DB1_SalidasExterioresDeMesa".Mesa[#Mesa].VelocidadLenta_E1E3 )
   END_RUNG
   RUNG wire#powerrail
      Contact( #Mx_ET10 )
   END_RUNG wire#w1
   RUNG wire#powerrail
      Contact( #Mx_ET11 )
   END_RUNG wire#w1
   RUNG wire#powerrail
      Contact( #Mx_ET12 )
   END_RUNG wire#w1
   RUNG wire#powerrail
      Contact( #Mx_ET02ESPERA )
   END_RUNG wire#w2
   RUNG wire#powerrail
      Contact( #Mx_VelocidadLenta_In )
   END_RUNG wire#w2
   RUNG wire#powerrail
      Contact( #EstadoZona.Manual_CBx )
   END_RUNG wire#w2
   // the same network as SCL:
   "DB1_SalidasExterioresDeMesa".Mesa[#Mesa].VelocidadLenta_E1E3 := ((#Mx_ET10Previo OR #Mx_ET10 OR #Mx_ET11 OR #Mx_ET12) AND (#CNTSeg_pHsMx.CVU >= #V_CNT_PasoLenta)) OR #Mx_ET02ESPERA OR #Mx_VelocidadLenta_In OR #EstadoZona.Manual_CBx;
END_REGION

REGION Network 71: SALIDAS - Sacar Centrador - COMPACTAR LA CARGA
   RUNG wire#powerrail
      Contact( #Mx_ET02 )
      Contact( #OrdSal_S00 )
      Contact( #OrdSalida_OK )
      Contact( #pHsMx_Seg )
      I_Contact( #CargaCompactada )
      Contact( #EstadoZona.Marcha_CBx )
      I_Contact( #EstadoVI.Error_Mx )
      I_Contact( #Error_Tx )
      Contact( #CIMCORP_MoveOK )
      Contact( #CIMCORP_OK )
      Coil( #MA_SacarCentrador )
   END_RUNG
   // the same network as SCL:
   #MA_SacarCentrador := #Mx_ET02 AND #OrdSal_S00 AND #OrdSalida_OK AND #pHsMx_Seg AND NOT #CargaCompactada AND #EstadoZona.Marcha_CBx AND NOT #EstadoVI.Error_Mx AND NOT #Error_Tx AND #CIMCORP_MoveOK AND #CIMCORP_OK;
END_REGION

REGION Network 72: SALIDAS - Recoger Centrador - DESCOMPACTAR LA CARGA
   RUNG wire#powerrail
      Contact( #Mx_ET02 )
      Contact( #OrdSal_S00 )
      Contact( #OrdSalida_OK )
      Contact( #CargaCompactada )
      I_Contact( #Centrador_OUT )
      Contact( #EstadoZona.Marcha_CBx )
      I_Contact( #EstadoVI.Error_Mx )
      I_Contact( #Error_Tx )
      Contact( #CIMCORP_MoveOK )
      Contact( #CIMCORP_OK )
      Coil( #MA_RecogerCentrador )
   END_RUNG
   // the same network as SCL:
   #MA_RecogerCentrador := #Mx_ET02 AND #OrdSal_S00 AND #OrdSalida_OK AND #CargaCompactada AND NOT #Centrador_OUT AND #EstadoZona.Marcha_CBx AND NOT #EstadoVI.Error_Mx AND NOT #Error_Tx AND #CIMCORP_MoveOK AND #CIMCORP_OK;
END_REGION

REGION Network 73: ESTADOS DE LA MESA
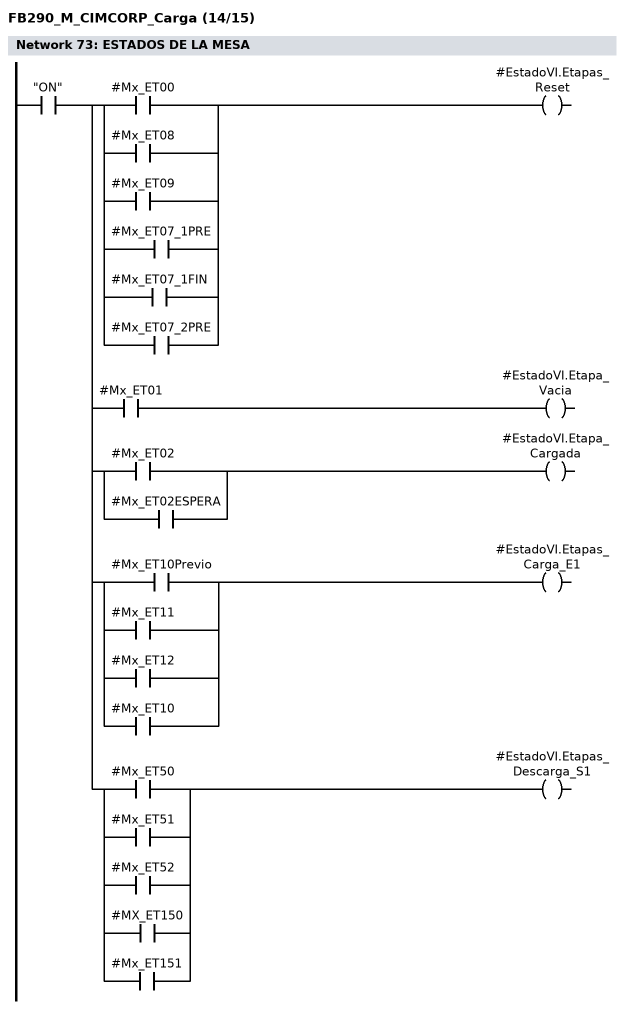
   RUNG wire#powerrail
      Contact( "ON" )
      wire#w1
      Contact( #Mx_ET00 )
      wire#w2
      Coil( #EstadoVI.Etapas_Reset )
   END_RUNG
   RUNG wire#w1
      Contact( #Mx_ET08 )
   END_RUNG wire#w2
   RUNG wire#w1
      Contact( #Mx_ET09 )
   END_RUNG wire#w2
   RUNG wire#w1
      Contact( #Mx_ET07_1PRE )
   END_RUNG wire#w2
   RUNG wire#w1
      Contact( #Mx_ET07_1FIN )
   END_RUNG wire#w2
   RUNG wire#w1
      Contact( #Mx_ET07_2PRE )
   END_RUNG wire#w2
   RUNG wire#w1
      Contact( #Mx_ET01 )
      Coil( #EstadoVI.Etapa_Vacia )
   END_RUNG
   RUNG wire#w1
      Contact( #Mx_ET02 )
      wire#w3
      Coil( #EstadoVI.Etapa_Cargada )
   END_RUNG
   RUNG wire#w1
      Contact( #Mx_ET02ESPERA )
   END_RUNG wire#w3
   RUNG wire#w1
      Contact( #Mx_ET10Previo )
      wire#w4
      Coil( #EstadoVI.Etapas_Carga_E1 )
   END_RUNG
   RUNG wire#w1
      Contact( #Mx_ET11 )
   END_RUNG wire#w4
   RUNG wire#w1
      Contact( #Mx_ET12 )
   END_RUNG wire#w4
   RUNG wire#w1
      Contact( #Mx_ET10 )
   END_RUNG wire#w4
   RUNG wire#w1
      Contact( #Mx_ET50 )
      wire#w5
      Coil( #EstadoVI.Etapas_Descarga_S1 )
   END_RUNG
   RUNG wire#w1
      Contact( #Mx_ET51 )
   END_RUNG wire#w5
   RUNG wire#w1
      Contact( #Mx_ET52 )
   END_RUNG wire#w5
   RUNG wire#w1
      Contact( #MX_ET150 )
   END_RUNG wire#w5
   RUNG wire#w1
      Contact( #Mx_ET151 )
   END_RUNG wire#w5
   // the same network as SCL:
   #EstadoVI.Etapas_Reset := "ON" AND (#Mx_ET00 OR #Mx_ET08 OR #Mx_ET09 OR #Mx_ET07_1PRE OR #Mx_ET07_1FIN OR #Mx_ET07_2PRE);
   #EstadoVI.Etapa_Vacia := "ON" AND #Mx_ET01;
   #EstadoVI.Etapa_Cargada := "ON" AND (#Mx_ET02 OR #Mx_ET02ESPERA);
   #EstadoVI.Etapas_Carga_E1 := "ON" AND (#Mx_ET10Previo OR #Mx_ET11 OR #Mx_ET12 OR #Mx_ET10);
   #EstadoVI.Etapas_Descarga_S1 := "ON" AND (#Mx_ET50 OR #Mx_ET51 OR #Mx_ET52 OR #MX_ET150 OR #Mx_ET151);
END_REGION

REGION Network 74: ENTRADAS DE LA MESA
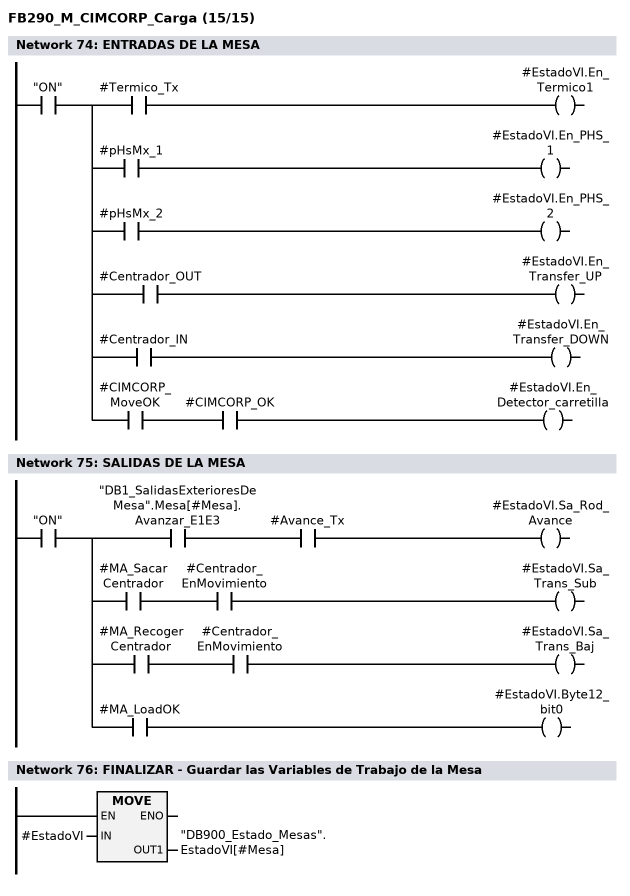
   RUNG wire#powerrail
      Contact( "ON" )
      wire#w1
      Contact( #Termico_Tx )
      Coil( #EstadoVI.En_Termico1 )
   END_RUNG
   RUNG wire#w1
      Contact( #pHsMx_1 )
      Coil( #EstadoVI.En_PHS_1 )
   END_RUNG
   RUNG wire#w1
      Contact( #pHsMx_2 )
      Coil( #EstadoVI.En_PHS_2 )
   END_RUNG
   RUNG wire#w1
      Contact( #Centrador_OUT )
      Coil( #EstadoVI.En_Transfer_UP )
   END_RUNG
   RUNG wire#w1
      Contact( #Centrador_IN )
      Coil( #EstadoVI.En_Transfer_DOWN )
   END_RUNG
   RUNG wire#w1
      Contact( #CIMCORP_MoveOK )
      Contact( #CIMCORP_OK )
      Coil( #EstadoVI.En_Detector_carretilla )
   END_RUNG
   // the same network as SCL:
   #EstadoVI.En_Termico1 := "ON" AND #Termico_Tx;
   #EstadoVI.En_PHS_1 := "ON" AND #pHsMx_1;
   #EstadoVI.En_PHS_2 := "ON" AND #pHsMx_2;
   #EstadoVI.En_Transfer_UP := "ON" AND #Centrador_OUT;
   #EstadoVI.En_Transfer_DOWN := "ON" AND #Centrador_IN;
   #EstadoVI.En_Detector_carretilla := "ON" AND #CIMCORP_MoveOK AND #CIMCORP_OK;
END_REGION

REGION Network 75: SALIDAS DE LA MESA
   RUNG wire#powerrail
      Contact( "ON" )
      wire#w1
      Contact( "DB1_SalidasExterioresDeMesa".Mesa[#Mesa].Avanzar_E1E3 )
      Contact( #Avance_Tx )
      Coil( #EstadoVI.Sa_Rod_Avance )
   END_RUNG
   RUNG wire#w1
      Contact( #MA_SacarCentrador )
      Contact( #Centrador_EnMovimiento )
      Coil( #EstadoVI.Sa_Trans_Sub )
   END_RUNG
   RUNG wire#w1
      Contact( #MA_RecogerCentrador )
      Contact( #Centrador_EnMovimiento )
      Coil( #EstadoVI.Sa_Trans_Baj )
   END_RUNG
   RUNG wire#w1
      Contact( #MA_LoadOK )
      Coil( #EstadoVI.Byte12_bit0 )
   END_RUNG
   // the same network as SCL:
   #EstadoVI.Sa_Rod_Avance := "ON" AND "DB1_SalidasExterioresDeMesa".Mesa[#Mesa].Avanzar_E1E3 AND #Avance_Tx;
   #EstadoVI.Sa_Trans_Sub := "ON" AND #MA_SacarCentrador AND #Centrador_EnMovimiento;
   #EstadoVI.Sa_Trans_Baj := "ON" AND #MA_RecogerCentrador AND #Centrador_EnMovimiento;
   #EstadoVI.Byte12_bit0 := "ON" AND #MA_LoadOK;
END_REGION

REGION Network 76: FINALIZAR - Guardar las Variables de Trabajo de la Mesa
   RUNG wire#powerrail
      Move(in := #EstadoVI, out1 => "DB900_Estado_Mesas".EstadoVI[#Mesa])
   END_RUNG
   // the same network as SCL:
   "DB900_Estado_Mesas".EstadoVI[#Mesa] := #EstadoVI;
END_REGION
END_FUNCTION_BLOCK
